LIN {X 0,Y 632.972,Z 1080.137,A -85,B 0,C 180,E1 6544.862,E2 6544.862} C_VEL
LIN {X 0,Y 629.315,Z 1123.898,A -85,B 0,C 180,E1 6550.738,E2 6550.738} C_VEL
LIN {X 0,Y 627.45,Z 1154.06,A -85,B 0,C 180,E1 6556.727,E2 6556.727} C_VEL
LIN {X 0,Y 627.035,Z 1171.451,A -85,B 0,C 180,E1 6562.357,E2 6562.357} C_VEL
LIN {X 0,Y 626.816,Z 1179.339,A -85,B 0,C 180,E1 6567.922,E2 6567.922} C_VEL
LIN {X 0,Y 626.99,Z 1178.178,A -85,B 0,C 180,E1 6573.468,E2 6573.468} C_VEL
LIN {X 0,Y 627.101,Z 1167.787,A -85,B 0,C 180,E1 6579.045,E2 6579.045} C_VEL
LIN {X 0,Y 627.936,Z 1145.964,A -85,B 0,C 180,E1 6585.071,E2 6585.071} C_VEL
LIN {X 0,Y 630.384,Z 1109.697,A -85,B 0,C 180,E1 6591.339,E2 6591.339} C_VEL
LIN {X 0,Y 634.84,Z 1059.626,A -85,B 0,C 180,E1 6597.186,E2 6597.186} C_VEL
LIN {X 0,Y 640.935,Z 997.311,A -85,B 0,C 180,E1 6602.167,E2 6602.167} C_VEL
LIN {X 0,Y 646.827,Z 930.309,A -85,B 0,C 180,E1 6605.71,E2 6605.71} C_VEL
LIN {X 0,Y 651.3,Z 859.749,A -85,B 0,C 180,E1 6607.946,E2 6607.946} C_VEL
LIN {X 0,Y 651.243,Z 808.043,A -85,B 0,C 180,E1 6608.958,E2 6608.958} C_VEL
LIN {X 0,Y 625.945,Z 762.06,A -85,B 0,C 180,E1 6612.013,E2 6612.013} C_VEL
LIN {X 0,Y 626.103,Z 762.06,A -85,B 0,C 180,E1 6620.047,E2 6620.047} C_VEL
LIN {X 0,Y 626.399,Z 762.06,A -85,B 0,C 180,E1 6628.62,E2 6628.62} C_VEL
LIN {X 0,Y 626.558,Z 762.06,A -85,B 0,C 180,E1 6637.961,E2 6637.961} C_VEL
LIN {X 0,Y 627.231,Z 762.06,A -85,B 0,C 180,E1 6646.724,E2 6646.724} C_VEL
LIN {X 0,Y 627.296,Z 762.06,A -85,B 0,C 180,E1 6656.747,E2 6656.747} C_VEL
LIN {X 0,Y 626.777,Z 762.06,A -85,B 0,C 180,E1 6666.27,E2 6666.27} C_VEL
LIN {X 0,Y 626.418,Z 762.06,A -85,B 0,C 180,E1 6674.754,E2 6674.754} C_VEL
LIN {X 0,Y 626.309,Z 762.06,A -85,B 0,C 180,E1 6682.078,E2 6682.078} C_VEL
LIN {X 0,Y 626.181,Z 762.06,A -85,B 0,C 180,E1 6690.708,E2 6690.708} C_VEL
LIN {X 0,Y 625.995,Z 762.06,A -85,B 0,C 180,E1 6698.209,E2 6698.209} C_VEL
LIN {X 0,Y 626.116,Z 762.06,A -85,B 0,C 180,E1 6703.678,E2 6703.678} C_VEL
LIN {X 0,Y 627.821,Z 770.775,A -85,B 0,C 180,E1 6704.212,E2 6704.212} C_VEL
LIN {X 0,Y 629.865,Z 783.636,A -85,B 0,C 180,E1 6704.574,E2 6704.574} C_VEL
LIN {X 0,Y 651.231,Z 823.405,A -85,B 0,C 180,E1 6706.95,E2 6706.95} C_VEL
LIN {X 0,Y 647.22,Z 901.729,A -85,B 0,C 180,E1 6708.805,E2 6708.805} C_VEL
LIN {X 0,Y 640.811,Z 974.236,A -85,B 0,C 180,E1 6711.939,E2 6711.939} C_VEL
LIN {X 0,Y 633.348,Z 1041.271,A -85,B 0,C 180,E1 6716.376,E2 6716.376} C_VEL
LIN {X 0,Y 626.505,Z 1100.933,A -85,B 0,C 180,E1 6722.094,E2 6722.094} C_VEL
LIN {X 0,Y 621.948,Z 1147.2,A -85,B 0,C 180,E1 6728.406,E2 6728.406} C_VEL
LIN {X 0,Y 619.779,Z 1179.297,A -85,B 0,C 180,E1 6734.748,E2 6734.748} C_VEL
LIN {X 0,Y 619.01,Z 1199.023,A -85,B 0,C 180,E1 6740.836,E2 6740.836} C_VEL
LIN {X 0,Y 618.831,Z 1208.374,A -85,B 0,C 180,E1 6746.486,E2 6746.486} C_VEL
LIN {X 0,Y 618.753,Z 1209.405,A -85,B 0,C 180,E1 6752.105,E2 6752.105} C_VEL
LIN {X 0,Y 618.943,Z 1202.167,A -85,B 0,C 180,E1 6757.743,E2 6757.743} C_VEL
LIN {X 0,Y 619.523,Z 1184.044,A -85,B 0,C 180,E1 6764.028,E2 6764.028} C_VEL
LIN {X 0,Y 621.435,Z 1154.124,A -85,B 0,C 180,E1 6770.425,E2 6770.425} C_VEL
LIN {X 0,Y 625.556,Z 1110.358,A -85,B 0,C 180,E1 6776.797,E2 6776.797} C_VEL
LIN {X 0,Y 632.02,Z 1052.823,A -85,B 0,C 180,E1 6782.674,E2 6782.674} C_VEL
LIN {X 0,Y 639.533,Z 985.869,A -85,B 0,C 180,E1 6787.417,E2 6787.417} C_VEL
LIN {X 0,Y 646.407,Z 914.616,A -85,B 0,C 180,E1 6790.745,E2 6790.745} C_VEL
LIN {X 0,Y 650.861,Z 841.464,A -85,B 0,C 180,E1 6792.732,E2 6792.732} C_VEL
LIN {X 0,Y 650.149,Z 816.893,A -85,B 0,C 180,E1 6793.253,E2 6793.253} C_VEL
LIN {X 0,Y 618.02,Z 762.06,A -85,B 0,C 180,E1 6796.943,E2 6796.943} C_VEL
LIN {X 0,Y 618.577,Z 762.06,A -85,B 0,C 180,E1 6805.212,E2 6805.212} C_VEL
LIN {X 0,Y 618.386,Z 762.06,A -85,B 0,C 180,E1 6814.546,E2 6814.546} C_VEL
LIN {X 0,Y 618.44,Z 762.06,A -85,B 0,C 180,E1 6823.591,E2 6823.591} C_VEL
LIN {X 0,Y 618.436,Z 762.06,A -85,B 0,C 180,E1 6832.228,E2 6832.228} C_VEL
LIN {X 0,Y 618.578,Z 762.06,A -85,B 0,C 180,E1 6839.283,E2 6839.283} C_VEL
LIN {X 0,Y 618.573,Z 762.06,A -85,B 0,C 180,E1 6846.839,E2 6846.839} C_VEL
LIN {X 0,Y 618.354,Z 762.06,A -85,B 0,C 180,E1 6854.921,E2 6854.921} C_VEL
LIN {X 0,Y 618.049,Z 762.06,A -85,B 0,C 180,E1 6863.057,E2 6863.057} C_VEL
LIN {X 0,Y 618.489,Z 762.06,A -85,B 0,C 180,E1 6871.828,E2 6871.828} C_VEL
LIN {X 0,Y 618.3,Z 762.06,A -85,B 0,C 180,E1 6880.562,E2 6880.562} C_VEL
LIN {X 0,Y 618.305,Z 763.681,A -85,B 0,C 180,E1 6887.36,E2 6887.36} C_VEL
LIN {X 0,Y 646.36,Z 813.844,A -85,B 0,C 180,E1 6890.637,E2 6890.637} C_VEL
LIN {X 0,Y 643.451,Z 889.072,A -85,B 0,C 180,E1 6892.263,E2 6892.263} C_VEL
LIN {X 0,Y 637.631,Z 960.527,A -85,B 0,C 180,E1 6895.184,E2 6895.184} C_VEL
LIN {X 0,Y 631.001,Z 1026.212,A -85,B 0,C 180,E1 6899.431,E2 6899.431} C_VEL
LIN {X 0,Y 625.13,Z 1083.1,A -85,B 0,C 180,E1 6904.88,E2 6904.88} C_VEL
LIN {X 0,Y 621.285,Z 1126.643,A -85,B 0,C 180,E1 6910.947,E2 6910.947} C_VEL
LIN {X 0,Y 619.446,Z 1155.409,A -85,B 0,C 180,E1 6916.913,E2 6916.913} C_VEL
LIN {X 0,Y 619.059,Z 1171.45,A -85,B 0,C 180,E1 6922.258,E2 6922.258} C_VEL
LIN {X 0,Y 618.82,Z 1179.339,A -85,B 0,C 180,E1 6927.895,E2 6927.895} C_VEL
LIN {X 0,Y 618.985,Z 1178.179,A -85,B 0,C 180,E1 6933.513,E2 6933.513} C_VEL
LIN {X 0,Y 619.092,Z 1165.857,A -85,B 0,C 180,E1 6939.875,E2 6939.875} C_VEL
LIN {X 0,Y 620.14,Z 1142.599,A -85,B 0,C 180,E1 6945.97,E2 6945.97} C_VEL
LIN {X 0,Y 622.856,Z 1107.043,A -85,B 0,C 180,E1 6951.985,E2 6951.985} C_VEL
LIN {X 0,Y 627.83,Z 1055.791,A -85,B 0,C 180,E1 6957.906,E2 6957.906} C_VEL
LIN {X 0,Y 634.324,Z 993.783,A -85,B 0,C 180,E1 6962.802,E2 6962.802} C_VEL
LIN {X 0,Y 640.691,Z 925.524,A -85,B 0,C 180,E1 6966.333,E2 6966.333} C_VEL
LIN {X 0,Y 645.573,Z 856.303,A -85,B 0,C 180,E1 6968.501,E2 6968.501} C_VEL
LIN {X 0,Y 645.401,Z 811.288,A -85,B 0,C 180,E1 6969.39,E2 6969.39} C_VEL
LIN {X 0,Y 617.998,Z 762.06,A -85,B 0,C 180,E1 6972.732,E2 6972.732} C_VEL
LIN {X 0,Y 618.138,Z 762.06,A -85,B 0,C 180,E1 6981.253,E2 6981.253} C_VEL
LIN {X 0,Y 618.383,Z 762.06,A -85,B 0,C 180,E1 6990.531,E2 6990.531} C_VEL
LIN {X 0,Y 618.488,Z 762.06,A -85,B 0,C 180,E1 6999.171,E2 6999.171} C_VEL
LIN {X 0,Y 619.321,Z 762.06,A -85,B 0,C 180,E1 7007.991,E2 7007.991} C_VEL
LIN {X 0,Y 619.217,Z 762.06,A -85,B 0,C 180,E1 7017.907,E2 7017.907} C_VEL
LIN {X 0,Y 618.579,Z 762.06,A -85,B 0,C 180,E1 7026.819,E2 7026.819} C_VEL
LIN {X 0,Y 618.378,Z 762.06,A -85,B 0,C 180,E1 7034.95,E2 7034.95} C_VEL
LIN {X 0,Y 618.109,Z 762.06,A -85,B 0,C 180,E1 7043.063,E2 7043.063} C_VEL
LIN {X 0,Y 618.003,Z 762.06,A -85,B 0,C 180,E1 7051.89,E2 7051.89} C_VEL
LIN {X 0,Y 617.716,Z 762.06,A -85,B 0,C 180,E1 7060.646,E2 7060.646} C_VEL
LIN {X 0,Y 618.142,Z 763.584,A -85,B 0,C 180,E1 7063.287,E2 7063.287} C_VEL
LIN {X 0,Y 629.865,Z 783.636,A -85,B 0,C 180,E1 7064.574,E2 7064.574} C_VEL
LIN {X 0,Y 640.224,Z 814.553,A -85,B 0,C 180,E1 7065.868,E2 7065.868} C_VEL
LIN {X 0,Y 645.268,Z 827.537,A -85,B 0,C 180,E1 7066.528,E2 7066.528} C_VEL
LIN {X 0,Y 640.734,Z 906.147,A -85,B 0,C 180,E1 7068.474,E2 7068.474} C_VEL
LIN {X 0,Y 633.667,Z 980.13,A -85,B 0,C 180,E1 7071.809,E2 7071.809} C_VEL
LIN {X 0,Y 625.559,Z 1048.266,A -85,B 0,C 180,E1 7076.534,E2 7076.534} C_VEL
LIN {X 0,Y 618.451,Z 1107.346,A -85,B 0,C 180,E1 7082.492,E2 7082.492} C_VEL
LIN {X 0,Y 614.002,Z 1153.543,A -85,B 0,C 180,E1 7089.215,E2 7089.215} C_VEL
LIN {X 0,Y 612.007,Z 1186.192,A -85,B 0,C 180,E1 7096.383,E2 7096.383} C_VEL
LIN {X 0,Y 611.482,Z 1204.733,A -85,B 0,C 180,E1 7103.591,E2 7103.591} C_VEL
LIN {X 0,Y 611.017,Z 1209.838,A -85,B 0,C 180,E1 7110.71,E2 7110.71} C_VEL
LIN {X 0,Y 610.986,Z 1203.526,A -85,B 0,C 180,E1 7117.128,E2 7117.128} C_VEL
LIN {X 0,Y 611.464,Z 1187.527,A -85,B 0,C 180,E1 7123.261,E2 7123.261} C_VEL
LIN {X 0,Y 613.202,Z 1159.147,A -85,B 0,C 180,E1 7129.766,E2 7129.766} C_VEL
LIN {X 0,Y 617.273,Z 1117.563,A -85,B 0,C 180,E1 7136.222,E2 7136.222} C_VEL
LIN {X 0,Y 624.02,Z 1060.465,A -85,B 0,C 180,E1 7142.405,E2 7142.405} C_VEL
LIN {X 0,Y 632.018,Z 994.245,A -85,B 0,C 180,E1 7147.364,E2 7147.364} C_VEL
LIN {X 0,Y 639.415,Z 923.76,A -85,B 0,C 180,E1 7150.864,E2 7150.864} C_VEL
LIN {X 0,Y 644.561,Z 848.588,A -85,B 0,C 180,E1 7153.084,E2 7153.084} C_VEL
LIN {X 0,Y 644.019,Z 819.648,A -85,B 0,C 180,E1 7153.719,E2 7153.719} C_VEL
LIN {X 0,Y 610.073,Z 762.06,A -85,B 0,C 180,E1 7157.493,E2 7157.493} C_VEL
LIN {X 0,Y 610.558,Z 762.06,A -85,B 0,C 180,E1 7166.31,E2 7166.31} C_VEL
LIN {X 0,Y 610.263,Z 762.06,A -85,B 0,C 180,E1 7175.095,E2 7175.095} C_VEL
LIN {X 0,Y 610.44,Z 762.06,A -85,B 0,C 180,E1 7183.37,E2 7183.37} C_VEL
LIN {X 0,Y 610.446,Z 762.06,A -85,B 0,C 180,E1 7192.125,E2 7192.125} C_VEL
LIN {X 0,Y 610.579,Z 762.06,A -85,B 0,C 180,E1 7199.273,E2 7199.273} C_VEL
LIN {X 0,Y 610.725,Z 762.06,A -85,B 0,C 180,E1 7206.406,E2 7206.406} C_VEL
LIN {X 0,Y 610.3,Z 762.06,A -85,B 0,C 180,E1 7215.122,E2 7215.122} C_VEL
LIN {X 0,Y 610.129,Z 762.06,A -85,B 0,C 180,E1 7222.665,E2 7222.665} C_VEL
LIN {X 0,Y 610.454,Z 762.06,A -85,B 0,C 180,E1 7231.015,E2 7231.015} C_VEL
LIN {X 0,Y 610.262,Z 762.06,A -85,B 0,C 180,E1 7239.343,E2 7239.343} C_VEL
LIN {X 0,Y 610.277,Z 763.855,A -85,B 0,C 180,E1 7246.599,E2 7246.599} C_VEL
LIN {X 0,Y 640.61,Z 817.11,A -85,B 0,C 180,E1 7250.202,E2 7250.202} C_VEL
LIN {X 0,Y 637.307,Z 890.904,A -85,B 0,C 180,E1 7251.834,E2 7251.834} C_VEL
LIN {X 0,Y 630.91,Z 960.513,A -85,B 0,C 180,E1 7254.758,E2 7254.758} C_VEL
LIN {X 0,Y 623.825,Z 1026.845,A -85,B 0,C 180,E1 7259.098,E2 7259.098} C_VEL
LIN {X 0,Y 617.637,Z 1083.093,A -85,B 0,C 180,E1 7264.554,E2 7264.554} C_VEL
LIN {X 0,Y 613.482,Z 1126.638,A -85,B 0,C 180,E1 7270.695,E2 7270.695} C_VEL
LIN {X 0,Y 611.529,Z 1155.408,A -85,B 0,C 180,E1 7276.74,E2 7276.74} C_VEL
LIN {X 0,Y 611.029,Z 1173.317,A -85,B 0,C 180,E1 7283.016,E2 7283.016} C_VEL
LIN {X 0,Y 610.859,Z 1179.847,A -85,B 0,C 180,E1 7289.29,E2 7289.29} C_VEL
LIN {X 0,Y 611.275,Z 1175.345,A -85,B 0,C 180,E1 7295.697,E2 7295.697} C_VEL
LIN {X 0,Y 612.229,Z 1156.406,A -85,B 0,C 180,E1 7302.883,E2 7302.883} C_VEL
LIN {X 0,Y 614.178,Z 1122.729,A -85,B 0,C 180,E1 7309.866,E2 7309.866} C_VEL
LIN {X 0,Y 618.595,Z 1076.123,A -85,B 0,C 180,E1 7316.154,E2 7316.154} C_VEL
LIN {X 0,Y 624.868,Z 1018.535,A -85,B 0,C 180,E1 7321.454,E2 7321.454} C_VEL
LIN {X 0,Y 631.781,Z 951.617,A -85,B 0,C 180,E1 7325.604,E2 7325.604} C_VEL
LIN {X 0,Y 637.934,Z 879.426,A -85,B 0,C 180,E1 7328.425,E2 7328.425} C_VEL
LIN {X 0,Y 639.65,Z 814.585,A -85,B 0,C 180,E1 7329.828,E2 7329.828} C_VEL
LIN {X 0,Y 610.11,Z 762.06,A -85,B 0,C 180,E1 7333.577,E2 7333.577} C_VEL
LIN {X 0,Y 610.17,Z 762.06,A -85,B 0,C 180,E1 7342.469,E2 7342.469} C_VEL
LIN {X 0,Y 610.341,Z 762.06,A -85,B 0,C 180,E1 7351.009,E2 7351.009} C_VEL
LIN {X 0,Y 610.46,Z 762.06,A -85,B 0,C 180,E1 7358.884,E2 7358.884} C_VEL
LIN {X 0,Y 611.247,Z 762.06,A -85,B 0,C 180,E1 7368.529,E2 7368.529} C_VEL
LIN {X 0,Y 611.236,Z 762.06,A -85,B 0,C 180,E1 7377.88,E2 7377.88} C_VEL
LIN {X 0,Y 610.707,Z 762.06,A -85,B 0,C 180,E1 7386.436,E2 7386.436} C_VEL
LIN {X 0,Y 610.321,Z 762.06,A -85,B 0,C 180,E1 7395.152,E2 7395.152} C_VEL
LIN {X 0,Y 610.181,Z 762.06,A -85,B 0,C 180,E1 7402.694,E2 7402.694} C_VEL
LIN {X 0,Y 610.098,Z 762.06,A -85,B 0,C 180,E1 7410.953,E2 7410.953} C_VEL
LIN {X 0,Y 609.786,Z 762.06,A -85,B 0,C 180,E1 7419.418,E2 7419.418} C_VEL
LIN {X 0,Y 610.156,Z 764.104,A -85,B 0,C 180,E1 7422.596,E2 7422.596} C_VEL
LIN {X 0,Y 640.224,Z 814.553,A -85,B 0,C 180,E1 7425.868,E2 7425.868} C_VEL
LIN {X 0,Y 639.91,Z 831.931,A -85,B 0,C 180,E1 7426.142,E2 7426.142} C_VEL
LIN {X 0,Y 639.001,Z 838.231,A -85,B 0,C 180,E1 7426.202,E2 7426.202} C_VEL
LIN {X 0,Y 633.48,Z 918.001,A -85,B 0,C 180,E1 7428.399,E2 7428.399} C_VEL
LIN {X 0,Y 625.961,Z 990.66,A -85,B 0,C 180,E1 7431.956,E2 7431.956} C_VEL
LIN {X 0,Y 617.597,Z 1056.725,A -85,B 0,C 180,E1 7436.844,E2 7436.844} C_VEL
LIN {X 0,Y 610.467,Z 1113.066,A -85,B 0,C 180,E1 7442.851,E2 7442.851} C_VEL
LIN {X 0,Y 605.973,Z 1157.974,A -85,B 0,C 180,E1 7449.76,E2 7449.76} C_VEL
LIN {X 0,Y 604.058,Z 1189.883,A -85,B 0,C 180,E1 7457.309,E2 7457.309} C_VEL
LIN {X 0,Y 603.382,Z 1205.908,A -85,B 0,C 180,E1 7464.249,E2 7464.249} C_VEL
LIN {X 0,Y 603.012,Z 1209.838,A -85,B 0,C 180,E1 7470.719,E2 7470.719} C_VEL
LIN {X 0,Y 602.988,Z 1203.524,A -85,B 0,C 180,E1 7477.223,E2 7477.223} C_VEL
LIN {X 0,Y 603.509,Z 1187.527,A -85,B 0,C 180,E1 7483.439,E2 7483.439} C_VEL
LIN {X 0,Y 605.336,Z 1160.03,A -85,B 0,C 180,E1 7489.861,E2 7489.861} C_VEL
LIN {X 0,Y 609.687,Z 1118.343,A -85,B 0,C 180,E1 7496.467,E2 7496.467} C_VEL
LIN {X 0,Y 616.724,Z 1062.438,A -85,B 0,C 180,E1 7502.64,E2 7502.64} C_VEL
LIN {X 0,Y 625.308,Z 995.453,A -85,B 0,C 180,E1 7507.748,E2 7507.748} C_VEL
LIN {X 0,Y 633.183,Z 924.545,A -85,B 0,C 180,E1 7511.317,E2 7511.317} C_VEL
LIN {X 0,Y 638.671,Z 849.436,A -85,B 0,C 180,E1 7513.559,E2 7513.559} C_VEL
LIN {X 0,Y 638.209,Z 823.006,A -85,B 0,C 180,E1 7514.158,E2 7514.158} C_VEL
LIN {X 0,Y 602.105,Z 762.06,A -85,B 0,C 180,E1 7518.367,E2 7518.367} C_VEL
LIN {X 0,Y 602.468,Z 762.06,A -85,B 0,C 180,E1 7527.186,E2 7527.186} C_VEL
LIN {X 0,Y 602.247,Z 762.06,A -85,B 0,C 180,E1 7535.412,E2 7535.412} C_VEL
LIN {X 0,Y 602.473,Z 762.06,A -85,B 0,C 180,E1 7543.143,E2 7543.143} C_VEL
LIN {X 0,Y 602.454,Z 762.06,A -85,B 0,C 180,E1 7552.02,E2 7552.02} C_VEL
LIN {X 0,Y 602.58,Z 762.06,A -85,B 0,C 180,E1 7559.264,E2 7559.264} C_VEL
LIN {X 0,Y 602.707,Z 762.06,A -85,B 0,C 180,E1 7566.492,E2 7566.492} C_VEL
LIN {X 0,Y 602.252,Z 762.06,A -85,B 0,C 180,E1 7575.329,E2 7575.329} C_VEL
LIN {X 0,Y 602.033,Z 762.06,A -85,B 0,C 180,E1 7583.161,E2 7583.161} C_VEL
LIN {X 0,Y 602.455,Z 762.06,A -85,B 0,C 180,E1 7591.078,E2 7591.078} C_VEL
LIN {X 0,Y 602.267,Z 762.06,A -85,B 0,C 180,E1 7599.969,E2 7599.969} C_VEL
LIN {X 0,Y 602.125,Z 762.964,A -85,B 0,C 180,E1 7605.782,E2 7605.782} C_VEL
LIN {X 0,Y 634.763,Z 820.076,A -85,B 0,C 180,E1 7609.742,E2 7609.742} C_VEL
LIN {X 0,Y 631.092,Z 894.25,A -85,B 0,C 180,E1 7611.45,E2 7611.45} C_VEL
LIN {X 0,Y 624.285,Z 962.539,A -85,B 0,C 180,E1 7614.396,E2 7614.396} C_VEL
LIN {X 0,Y 616.159,Z 1031.496,A -85,B 0,C 180,E1 7619.086,E2 7619.086} C_VEL
LIN {X 0,Y 609.691,Z 1087.332,A -85,B 0,C 180,E1 7624.72,E2 7624.72} C_VEL
LIN {X 0,Y 605.444,Z 1129.882,A -85,B 0,C 180,E1 7630.998,E2 7630.998} C_VEL
LIN {X 0,Y 603.483,Z 1158.086,A -85,B 0,C 180,E1 7637.299,E2 7637.299} C_VEL
LIN {X 0,Y 603.087,Z 1174.516,A -85,B 0,C 180,E1 7643.64,E2 7643.64} C_VEL
LIN {X 0,Y 602.857,Z 1179.847,A -85,B 0,C 180,E1 7649.281,E2 7649.281} C_VEL
LIN {X 0,Y 603.303,Z 1175.346,A -85,B 0,C 180,E1 7655.772,E2 7655.772} C_VEL
LIN {X 0,Y 604.272,Z 1156.407,A -85,B 0,C 180,E1 7663.055,E2 7663.055} C_VEL
LIN {X 0,Y 606.328,Z 1123.607,A -85,B 0,C 180,E1 7669.981,E2 7669.981} C_VEL
LIN {X 0,Y 611.098,Z 1076.452,A -85,B 0,C 180,E1 7676.463,E2 7676.463} C_VEL
LIN {X 0,Y 617.827,Z 1018.541,A -85,B 0,C 180,E1 7681.854,E2 7681.854} C_VEL
LIN {X 0,Y 625.884,Z 948.387,A -85,B 0,C 180,E1 7686.246,E2 7686.246} C_VEL
LIN {X 0,Y 632.245,Z 876.975,A -85,B 0,C 180,E1 7688.99,E2 7688.99} C_VEL
LIN {X 0,Y 633.798,Z 817.777,A -85,B 0,C 180,E1 7690.289,E2 7690.289} C_VEL
LIN {X 0,Y 602.12,Z 762.06,A -85,B 0,C 180,E1 7694.292,E2 7694.292} C_VEL
LIN {X 0,Y 602.142,Z 762.06,A -85,B 0,C 180,E1 7703.694,E2 7703.694} C_VEL
LIN {X 0,Y 602.259,Z 762.06,A -85,B 0,C 180,E1 7712.227,E2 7712.227} C_VEL
LIN {X 0,Y 602.323,Z 762.06,A -85,B 0,C 180,E1 7720.767,E2 7720.767} C_VEL
LIN {X 0,Y 603.225,Z 762.06,A -85,B 0,C 180,E1 7729.137,E2 7729.137} C_VEL
LIN {X 0,Y 603.233,Z 762.06,A -85,B 0,C 180,E1 7737.852,E2 7737.852} C_VEL
LIN {X 0,Y 602.676,Z 762.06,A -85,B 0,C 180,E1 7746.522,E2 7746.522} C_VEL
LIN {X 0,Y 602.279,Z 762.06,A -85,B 0,C 180,E1 7755.359,E2 7755.359} C_VEL
LIN {X 0,Y 602.071,Z 762.06,A -85,B 0,C 180,E1 7763.162,E2 7763.162} C_VEL
LIN {X 0,Y 602.091,Z 762.06,A -85,B 0,C 180,E1 7771.134,E2 7771.134} C_VEL
LIN {X 0,Y 601.736,Z 762.06,A -85,B 0,C 180,E1 7780.051,E2 7780.051} C_VEL
LIN {X 0,Y 601.924,Z 763.538,A -85,B 0,C 180,E1 7781.827,E2 7781.827} C_VEL
LIN {X 0,Y 639.368,Z 830.222,A -85,B 0,C 180,E1 7786.074,E2 7786.074} C_VEL
LIN {X 0,Y 639.001,Z 838.231,A -85,B 0,C 180,E1 7786.202,E2 7786.202} C_VEL
LIN {X 0,Y 631.54,Z 872.791,A -85,B 0,C 180,E1 7786.489,E2 7786.489} C_VEL
LIN {X 0,Y 624.788,Z 945.294,A -85,B 0,C 180,E1 7789.069,E2 7789.069} C_VEL
LIN {X 0,Y 615.988,Z 1016.482,A -85,B 0,C 180,E1 7793.185,E2 7793.185} C_VEL
LIN {X 0,Y 607.505,Z 1079.463,A -85,B 0,C 180,E1 7798.613,E2 7798.613} C_VEL
LIN {X 0,Y 600.829,Z 1132.474,A -85,B 0,C 180,E1 7805.188,E2 7805.188} C_VEL
LIN {X 0,Y 596.838,Z 1172.135,A -85,B 0,C 180,E1 7812.407,E2 7812.407} C_VEL
LIN {X 0,Y 595.351,Z 1195.465,A -85,B 0,C 180,E1 7819.049,E2 7819.049} C_VEL
LIN {X 0,Y 595.088,Z 1206.795,A -85,B 0,C 180,E1 7824.881,E2 7824.881} C_VEL
LIN {X 0,Y 595.032,Z 1209.838,A -85,B 0,C 180,E1 7830.729,E2 7830.729} C_VEL
LIN {X 0,Y 594.999,Z 1203.521,A -85,B 0,C 180,E1 7837.32,E2 7837.32} C_VEL
LIN {X 0,Y 595.591,Z 1186.203,A -85,B 0,C 180,E1 7843.997,E2 7843.997} C_VEL
LIN {X 0,Y 597.679,Z 1158.561,A -85,B 0,C 180,E1 7850.418,E2 7850.418} C_VEL
LIN {X 0,Y 602.303,Z 1116.951,A -85,B 0,C 180,E1 7857.009,E2 7857.009} C_VEL
LIN {X 0,Y 609.999,Z 1059.857,A -85,B 0,C 180,E1 7863.306,E2 7863.306} C_VEL
LIN {X 0,Y 619.009,Z 993.875,A -85,B 0,C 180,E1 7868.316,E2 7868.316} C_VEL
LIN {X 0,Y 627.143,Z 924.111,A -85,B 0,C 180,E1 7871.824,E2 7871.824} C_VEL
LIN {X 0,Y 632.814,Z 849.722,A -85,B 0,C 180,E1 7874.048,E2 7874.048} C_VEL
LIN {X 0,Y 632.259,Z 826.44,A -85,B 0,C 180,E1 7874.572,E2 7874.572} C_VEL
LIN {X 0,Y 594.208,Z 762.06,A -85,B 0,C 180,E1 7879.119,E2 7879.119} C_VEL
LIN {X 0,Y 594.409,Z 762.06,A -85,B 0,C 180,E1 7886.684,E2 7886.684} C_VEL
LIN {X 0,Y 594.237,Z 762.06,A -85,B 0,C 180,E1 7895.058,E2 7895.058} C_VEL
LIN {X 0,Y 594.259,Z 762.06,A -85,B 0,C 180,E1 7904.428,E2 7904.428} C_VEL
LIN {X 0,Y 594.462,Z 762.06,A -85,B 0,C 180,E1 7911.912,E2 7911.912} C_VEL
LIN {X 0,Y 594.593,Z 762.06,A -85,B 0,C 180,E1 7919.254,E2 7919.254} C_VEL
LIN {X 0,Y 594.67,Z 762.06,A -85,B 0,C 180,E1 7926.58,E2 7926.58} C_VEL
LIN {X 0,Y 594.213,Z 762.06,A -85,B 0,C 180,E1 7935.542,E2 7935.542} C_VEL
LIN {X 0,Y 594.01,Z 762.06,A -85,B 0,C 180,E1 7943.315,E2 7943.315} C_VEL
LIN {X 0,Y 594.429,Z 762.06,A -85,B 0,C 180,E1 7951.546,E2 7951.546} C_VEL
LIN {X 0,Y 594.18,Z 762.06,A -85,B 0,C 180,E1 7960.626,E2 7960.626} C_VEL
LIN {X 0,Y 594.256,Z 763.545,A -85,B 0,C 180,E1 7964.987,E2 7964.987} C_VEL
LIN {X 0,Y 629.008,Z 823.213,A -85,B 0,C 180,E1 7969.285,E2 7969.285} C_VEL
LIN {X 0,Y 625.064,Z 895.42,A -85,B 0,C 180,E1 7970.985,E2 7970.985} C_VEL
LIN {X 0,Y 617.855,Z 963.225,A -85,B 0,C 180,E1 7973.944,E2 7973.944} C_VEL
LIN {X 0,Y 609.218,Z 1030.33,A -85,B 0,C 180,E1 7978.589,E2 7978.589} C_VEL
LIN {X 0,Y 602.317,Z 1086.289,A -85,B 0,C 180,E1 7984.26,E2 7984.26} C_VEL
LIN {X 0,Y 597.641,Z 1129.879,A -85,B 0,C 180,E1 7990.74,E2 7990.74} C_VEL
LIN {X 0,Y 595.539,Z 1158.083,A -85,B 0,C 180,E1 7997.127,E2 7997.127} C_VEL
LIN {X 0,Y 595.039,Z 1174.288,A -85,B 0,C 180,E1 8003.416,E2 8003.416} C_VEL
LIN {X 0,Y 594.872,Z 1179.846,A -85,B 0,C 180,E1 8009.271,E2 8009.271} C_VEL
LIN {X 0,Y 595.331,Z 1175.399,A -85,B 0,C 180,E1 8015.819,E2 8015.819} C_VEL
LIN {X 0,Y 596.288,Z 1156.409,A -85,B 0,C 180,E1 8023.233,E2 8023.233} C_VEL
LIN {X 0,Y 598.52,Z 1123.609,A -85,B 0,C 180,E1 8030.253,E2 8030.253} C_VEL
LIN {X 0,Y 603.521,Z 1077.639,A -85,B 0,C 180,E1 8036.677,E2 8036.677} C_VEL
LIN {X 0,Y 610.673,Z 1019.813,A -85,B 0,C 180,E1 8042.167,E2 8042.167} C_VEL
LIN {X 0,Y 618.995,Z 953.671,A -85,B 0,C 180,E1 8046.473,E2 8046.473} C_VEL
LIN {X 0,Y 625.947,Z 882.027,A -85,B 0,C 180,E1 8049.353,E2 8049.353} C_VEL
LIN {X 0,Y 627.928,Z 820.81,A -85,B 0,C 180,E1 8050.766,E2 8050.766} C_VEL
LIN {X 0,Y 594.191,Z 762.06,A -85,B 0,C 180,E1 8055.133,E2 8055.133} C_VEL
LIN {X 0,Y 594.11,Z 762.06,A -85,B 0,C 180,E1 8064.931,E2 8064.931} C_VEL
LIN {X 0,Y 594.228,Z 762.06,A -85,B 0,C 180,E1 8073.466,E2 8073.466} C_VEL
LIN {X 0,Y 594.327,Z 762.06,A -85,B 0,C 180,E1 8081.4,E2 8081.4} C_VEL
LIN {X 0,Y 595.211,Z 762.06,A -85,B 0,C 180,E1 8088.989,E2 8088.989} C_VEL
LIN {X 0,Y 595.229,Z 762.06,A -85,B 0,C 180,E1 8097.823,E2 8097.823} C_VEL
LIN {X 0,Y 594.641,Z 762.06,A -85,B 0,C 180,E1 8106.611,E2 8106.611} C_VEL
LIN {X 0,Y 594.527,Z 762.06,A -85,B 0,C 180,E1 8114.051,E2 8114.051} C_VEL
LIN {X 0,Y 594.045,Z 762.06,A -85,B 0,C 180,E1 8123.347,E2 8123.347} C_VEL
LIN {X 0,Y 594.024,Z 762.06,A -85,B 0,C 180,E1 8131.605,E2 8131.605} C_VEL
LIN {X 0,Y 593.766,Z 762.06,A -85,B 0,C 180,E1 8138.83,E2 8138.83} C_VEL
LIN {X 0,Y 593.896,Z 763.614,A -85,B 0,C 180,E1 8141.039,E2 8141.039} C_VEL
LIN {X 0,Y 633.4,Z 831.798,A -85,B 0,C 180,E1 8145.61,E2 8145.61} C_VEL
LIN {X 0,Y 631.54,Z 872.791,A -85,B 0,C 180,E1 8146.489,E2 8146.489} C_VEL
LIN {X 0,Y 622.689,Z 906.696,A -85,B 0,C 180,E1 8147.015,E2 8147.015} C_VEL
LIN {X 0,Y 614.522,Z 979.053,A -85,B 0,C 180,E1 8150.32,E2 8150.32} C_VEL
LIN {X 0,Y 605.058,Z 1046.326,A -85,B 0,C 180,E1 8155.058,E2 8155.058} C_VEL
LIN {X 0,Y 596.431,Z 1105.461,A -85,B 0,C 180,E1 8161.142,E2 8161.142} C_VEL
LIN {X 0,Y 590.727,Z 1150.518,A -85,B 0,C 180,E1 8167.805,E2 8167.805} C_VEL
LIN {X 0,Y 587.977,Z 1182.006,A -85,B 0,C 180,E1 8174.626,E2 8174.626} C_VEL
LIN {X 0,Y 587.094,Z 1200.615,A -85,B 0,C 180,E1 8181.083,E2 8181.083} C_VEL
LIN {X 0,Y 587.153,Z 1209.403,A -85,B 0,C 180,E1 8187.778,E2 8187.778} C_VEL
LIN {X 0,Y 587.328,Z 1206.281,A -85,B 0,C 180,E1 8195.616,E2 8195.616} C_VEL
LIN {X 0,Y 587.539,Z 1191.036,A -85,B 0,C 180,E1 8202.672,E2 8202.672} C_VEL
LIN {X 0,Y 589.398,Z 1163.87,A -85,B 0,C 180,E1 8209.649,E2 8209.649} C_VEL
LIN {X 0,Y 594.118,Z 1123.159,A -85,B 0,C 180,E1 8216.53,E2 8216.53} C_VEL
LIN {X 0,Y 601.845,Z 1068.373,A -85,B 0,C 180,E1 8222.942,E2 8222.942} C_VEL
LIN {X 0,Y 611.221,Z 1003.832,A -85,B 0,C 180,E1 8228.159,E2 8228.159} C_VEL
LIN {X 0,Y 620.196,Z 933.124,A -85,B 0,C 180,E1 8231.963,E2 8231.963} C_VEL
LIN {X 0,Y 626.092,Z 859.422,A -85,B 0,C 180,E1 8234.324,E2 8234.324} C_VEL
LIN {X 0,Y 626.084,Z 829.765,A -85,B 0,C 180,E1 8235.002,E2 8235.002} C_VEL
LIN {X 0,Y 586.179,Z 762.06,A -85,B 0,C 180,E1 8239.796,E2 8239.796} C_VEL
LIN {X 0,Y 586.333,Z 762.06,A -85,B 0,C 180,E1 8247.931,E2 8247.931} C_VEL
LIN {X 0,Y 586.118,Z 762.06,A -85,B 0,C 180,E1 8256.707,E2 8256.707} C_VEL
LIN {X 0,Y 586.275,Z 762.06,A -85,B 0,C 180,E1 8264.211,E2 8264.211} C_VEL
LIN {X 0,Y 586.483,Z 762.06,A -85,B 0,C 180,E1 8271.801,E2 8271.801} C_VEL
LIN {X 0,Y 586.594,Z 762.06,A -85,B 0,C 180,E1 8279.244,E2 8279.244} C_VEL
LIN {X 0,Y 586.638,Z 762.06,A -85,B 0,C 180,E1 8286.671,E2 8286.671} C_VEL
LIN {X 0,Y 586.47,Z 762.06,A -85,B 0,C 180,E1 8294.217,E2 8294.217} C_VEL
LIN {X 0,Y 586.011,Z 762.06,A -85,B 0,C 180,E1 8303.269,E2 8303.269} C_VEL
LIN {X 0,Y 586.366,Z 762.06,A -85,B 0,C 180,E1 8312.031,E2 8312.031} C_VEL
LIN {X 0,Y 586.169,Z 762.06,A -85,B 0,C 180,E1 8321.302,E2 8321.302} C_VEL
LIN {X 0,Y 586.206,Z 763.284,A -85,B 0,C 180,E1 8324.126,E2 8324.126} C_VEL
LIN {X 0,Y 623.291,Z 826.304,A -85,B 0,C 180,E1 8328.818,E2 8328.818} C_VEL
LIN {X 0,Y 618.854,Z 898.927,A -85,B 0,C 180,E1 8330.587,E2 8330.587} C_VEL
LIN {X 0,Y 611.169,Z 966.822,A -85,B 0,C 180,E1 8333.651,E2 8333.651} C_VEL
LIN {X 0,Y 602.035,Z 1031.851,A -85,B 0,C 180,E1 8338.291,E2 8338.291} C_VEL
LIN {X 0,Y 594.653,Z 1087.887,A -85,B 0,C 180,E1 8344.106,E2 8344.106} C_VEL
LIN {X 0,Y 589.853,Z 1129.975,A -85,B 0,C 180,E1 8350.495,E2 8350.495} C_VEL
LIN {X 0,Y 587.602,Z 1158.08,A -85,B 0,C 180,E1 8356.95,E2 8356.95} C_VEL
LIN {X 0,Y 587.038,Z 1174.287,A -85,B 0,C 180,E1 8363.326,E2 8363.326} C_VEL
LIN {X 0,Y 586.871,Z 1179.846,A -85,B 0,C 180,E1 8369.261,E2 8369.261} C_VEL
LIN {X 0,Y 587.346,Z 1175.341,A -85,B 0,C 180,E1 8375.935,E2 8375.935} C_VEL
LIN {X 0,Y 588.301,Z 1156.411,A -85,B 0,C 180,E1 8383.416,E2 8383.416} C_VEL
LIN {X 0,Y 590.795,Z 1122.844,A -85,B 0,C 180,E1 8390.669,E2 8390.669} C_VEL
LIN {X 0,Y 596.156,Z 1076.419,A -85,B 0,C 180,E1 8397.185,E2 8397.185} C_VEL
LIN {X 0,Y 604.578,Z 1014.365,A -85,B 0,C 180,E1 8403.065,E2 8403.065} C_VEL
LIN {X 0,Y 613.379,Z 949.648,A -85,B 0,C 180,E1 8407.183,E2 8407.183} C_VEL
LIN {X 0,Y 620.384,Z 879.671,A -85,B 0,C 180,E1 8409.938,E2 8409.938} C_VEL
LIN {X 0,Y 622.12,Z 823.861,A -85,B 0,C 180,E1 8411.245,E2 8411.245} C_VEL
LIN {X 0,Y 586.081,Z 762.06,A -85,B 0,C 180,E1 8415.948,E2 8415.948} C_VEL
LIN {X 0,Y 586.095,Z 762.06,A -85,B 0,C 180,E1 8424.596,E2 8424.596} C_VEL
LIN {X 0,Y 586.194,Z 762.06,A -85,B 0,C 180,E1 8433.196,E2 8433.196} C_VEL
LIN {X 0,Y 586.298,Z 762.06,A -85,B 0,C 180,E1 8441.135,E2 8441.135} C_VEL
LIN {X 0,Y 587.241,Z 762.06,A -85,B 0,C 180,E1 8448.838,E2 8448.838} C_VEL
LIN {X 0,Y 587.224,Z 762.06,A -85,B 0,C 180,E1 8457.793,E2 8457.793} C_VEL
LIN {X 0,Y 586.627,Z 762.06,A -85,B 0,C 180,E1 8466.701,E2 8466.701} C_VEL
LIN {X 0,Y 586.473,Z 762.06,A -85,B 0,C 180,E1 8474.248,E2 8474.248} C_VEL
LIN {X 0,Y 586.061,Z 762.06,A -85,B 0,C 180,E1 8483.273,E2 8483.273} C_VEL
LIN {X 0,Y 585.937,Z 762.06,A -85,B 0,C 180,E1 8492.093,E2 8492.093} C_VEL
LIN {X 0,Y 585.758,Z 763.249,A -85,B 0,C 180,E1 8500.188,E2 8500.188} C_VEL
LIN {X 0,Y 627.244,Z 834.133,A -85,B 0,C 180,E1 8505.168,E2 8505.168} C_VEL
LIN {X 0,Y 622.689,Z 906.696,A -85,B 0,C 180,E1 8507.015,E2 8507.015} C_VEL
LIN {X 0,Y 614.028,Z 928.795,A -85,B 0,C 180,E1 8507.343,E2 8507.343} C_VEL
LIN {X 0,Y 605.269,Z 999.674,A -85,B 0,C 180,E1 8511.086,E2 8511.086} C_VEL
LIN {X 0,Y 595.428,Z 1064.977,A -85,B 0,C 180,E1 8516.303,E2 8516.303} C_VEL
LIN {X 0,Y 587.228,Z 1120.285,A -85,B 0,C 180,E1 8522.715,E2 8522.715} C_VEL
LIN {X 0,Y 582.141,Z 1163.606,A -85,B 0,C 180,E1 8530.042,E2 8530.042} C_VEL
LIN {X 0,Y 579.864,Z 1193.289,A -85,B 0,C 180,E1 8537.922,E2 8537.922} C_VEL
LIN {X 0,Y 579.164,Z 1206.789,A -85,B 0,C 180,E1 8544.74,E2 8544.74} C_VEL
LIN {X 0,Y 579.037,Z 1209.838,A -85,B 0,C 180,E1 8550.749,E2 8550.749} C_VEL
LIN {X 0,Y 579.006,Z 1203.516,A -85,B 0,C 180,E1 8557.523,E2 8557.523} C_VEL
LIN {X 0,Y 579.804,Z 1186.201,A -85,B 0,C 180,E1 8564.386,E2 8564.386} C_VEL
LIN {X 0,Y 582.454,Z 1155.592,A -85,B 0,C 180,E1 8571.576,E2 8571.576} C_VEL
LIN {X 0,Y 588.637,Z 1109.819,A -85,B 0,C 180,E1 8578.703,E2 8578.703} C_VEL
LIN {X 0,Y 597.479,Z 1051.475,A -85,B 0,C 180,E1 8584.955,E2 8584.955} C_VEL
LIN {X 0,Y 607.321,Z 985.398,A -85,B 0,C 180,E1 8589.812,E2 8589.812} C_VEL
LIN {X 0,Y 615.429,Z 918.9,A -85,B 0,C 180,E1 8593.011,E2 8593.011} C_VEL
LIN {X 0,Y 620.86,Z 846.059,A -85,B 0,C 180,E1 8595.073,E2 8595.073} C_VEL
LIN {X 0,Y 619.481,Z 832.28,A -85,B 0,C 180,E1 8595.493,E2 8595.493} C_VEL
LIN {X 0,Y 578.194,Z 762.06,A -85,B 0,C 180,E1 8600.688,E2 8600.688} C_VEL
LIN {X 0,Y 578.276,Z 762.06,A -85,B 0,C 180,E1 8609.197,E2 8609.197} C_VEL
LIN {X 0,Y 578.05,Z 762.06,A -85,B 0,C 180,E1 8617.604,E2 8617.604} C_VEL
LIN {X 0,Y 578.221,Z 762.06,A -85,B 0,C 180,E1 8625.544,E2 8625.544} C_VEL
LIN {X 0,Y 578.343,Z 762.06,A -85,B 0,C 180,E1 8633.202,E2 8633.202} C_VEL
LIN {X 0,Y 578.45,Z 762.06,A -85,B 0,C 180,E1 8640.736,E2 8640.736} C_VEL
LIN {X 0,Y 578.337,Z 762.06,A -85,B 0,C 180,E1 8648.284,E2 8648.284} C_VEL
LIN {X 0,Y 578.14,Z 762.06,A -85,B 0,C 180,E1 8656.784,E2 8656.784} C_VEL
LIN {X 0,Y 577.972,Z 762.06,A -85,B 0,C 180,E1 8665.66,E2 8665.66} C_VEL
LIN {X 0,Y 578.334,Z 762.06,A -85,B 0,C 180,E1 8674.332,E2 8674.332} C_VEL
LIN {X 0,Y 578.37,Z 764.01,A -85,B 0,C 180,E1 8683.269,E2 8683.269} C_VEL
LIN {X 0,Y 617.528,Z 829.414,A -85,B 0,C 180,E1 8688.339,E2 8688.339} C_VEL
LIN {X 0,Y 612.763,Z 901.876,A -85,B 0,C 180,E1 8690.162,E2 8690.162} C_VEL
LIN {X 0,Y 604.642,Z 969.043,A -85,B 0,C 180,E1 8693.265,E2 8693.265} C_VEL
LIN {X 0,Y 595.029,Z 1033.504,A -85,B 0,C 180,E1 8697.96,E2 8697.96} C_VEL
LIN {X 0,Y 586.554,Z 1092.338,A -85,B 0,C 180,E1 8704.339,E2 8704.339} C_VEL
LIN {X 0,Y 581.694,Z 1133.803,A -85,B 0,C 180,E1 8710.983,E2 8710.983} C_VEL
LIN {X 0,Y 579.545,Z 1160.579,A -85,B 0,C 180,E1 8717.534,E2 8717.534} C_VEL
LIN {X 0,Y 579.198,Z 1175.678,A -85,B 0,C 180,E1 8724.103,E2 8724.103} C_VEL
LIN {X 0,Y 579.469,Z 1179.824,A -85,B 0,C 180,E1 8730.751,E2 8730.751} C_VEL
LIN {X 0,Y 579.352,Z 1171.251,A -85,B 0,C 180,E1 8738.279,E2 8738.279} C_VEL
LIN {X 0,Y 580.245,Z 1150.802,A -85,B 0,C 180,E1 8745.132,E2 8745.132} C_VEL
LIN {X 0,Y 583.427,Z 1117.041,A -85,B 0,C 180,E1 8751.943,E2 8751.943} C_VEL
LIN {X 0,Y 589.685,Z 1068.827,A -85,B 0,C 180,E1 8758.411,E2 8758.411} C_VEL
LIN {X 0,Y 599.005,Z 1007.843,A -85,B 0,C 180,E1 8764.067,E2 8764.067} C_VEL
LIN {X 0,Y 608.249,Z 942.473,A -85,B 0,C 180,E1 8768.063,E2 8768.063} C_VEL
LIN {X 0,Y 615.342,Z 872.939,A -85,B 0,C 180,E1 8770.644,E2 8770.644} C_VEL
LIN {X 0,Y 616.568,Z 827.594,A -85,B 0,C 180,E1 8771.693,E2 8771.693} C_VEL
LIN {X 0,Y 578.021,Z 762.06,A -85,B 0,C 180,E1 8776.802,E2 8776.802} C_VEL
LIN {X 0,Y 578.048,Z 762.06,A -85,B 0,C 180,E1 8785.734,E2 8785.734} C_VEL
LIN {X 0,Y 578.242,Z 762.06,A -85,B 0,C 180,E1 8794.801,E2 8794.801} C_VEL
LIN {X 0,Y 578.652,Z 762.06,A -85,B 0,C 180,E1 8804.029,E2 8804.029} C_VEL
LIN {X 0,Y 578.584,Z 762.06,A -85,B 0,C 180,E1 8811.72,E2 8811.72} C_VEL
LIN {X 0,Y 578.633,Z 762.06,A -85,B 0,C 180,E1 8819.264,E2 8819.264} C_VEL
LIN {X 0,Y 578.593,Z 762.06,A -85,B 0,C 180,E1 8826.795,E2 8826.795} C_VEL
LIN {X 0,Y 578.412,Z 762.06,A -85,B 0,C 180,E1 8834.451,E2 8834.451} C_VEL
LIN {X 0,Y 578.127,Z 762.06,A -85,B 0,C 180,E1 8842.392,E2 8842.392} C_VEL
LIN {X 0,Y 577.948,Z 762.06,A -85,B 0,C 180,E1 8851.481,E2 8851.481} C_VEL
LIN {X 0,Y 577.914,Z 763.772,A -85,B 0,C 180,E1 8859.343,E2 8859.343} C_VEL
LIN {X 0,Y 621.043,Z 837.745,A -85,B 0,C 180,E1 8864.745,E2 8864.745} C_VEL
LIN {X 0,Y 615.263,Z 917.722,A -85,B 0,C 180,E1 8866.922,E2 8866.922} C_VEL
LIN {X 0,Y 614.028,Z 928.795,A -85,B 0,C 180,E1 8867.343,E2 8867.343} C_VEL
LIN {X 0,Y 604.257,Z 961.165,A -85,B 0,C 180,E1 8868.364,E2 8868.364} C_VEL
LIN {X 0,Y 594.44,Z 1027.751,A -85,B 0,C 180,E1 8872.6,E2 8872.6} C_VEL
LIN {X 0,Y 584.407,Z 1089.748,A -85,B 0,C 180,E1 8878.463,E2 8878.463} C_VEL
LIN {X 0,Y 576.91,Z 1139.778,A -85,B 0,C 180,E1 8885.316,E2 8885.316} C_VEL
LIN {X 0,Y 572.729,Z 1176.407,A -85,B 0,C 180,E1 8892.716,E2 8892.716} C_VEL
LIN {X 0,Y 571.232,Z 1198.062,A -85,B 0,C 180,E1 8899.635,E2 8899.635} C_VEL
LIN {X 0,Y 570.876,Z 1208.373,A -85,B 0,C 180,E1 8906.191,E2 8906.191} C_VEL
LIN {X 0,Y 570.819,Z 1209.405,A -85,B 0,C 180,E1 8912.282,E2 8912.282} C_VEL
LIN {X 0,Y 571.293,Z 1200.616,A -85,B 0,C 180,E1 8919.163,E2 8919.163} C_VEL
LIN {X 0,Y 573.129,Z 1177.815,A -85,B 0,C 180,E1 8926.908,E2 8926.908} C_VEL
LIN {X 0,Y 577.234,Z 1139.339,A -85,B 0,C 180,E1 8934.744,E2 8934.744} C_VEL
LIN {X 0,Y 584.721,Z 1088.293,A -85,B 0,C 180,E1 8941.699,E2 8941.699} C_VEL
LIN {X 0,Y 594.715,Z 1026.436,A -85,B 0,C 180,E1 8947.5,E2 8947.5} C_VEL
LIN {X 0,Y 604.145,Z 960.293,A -85,B 0,C 180,E1 8951.696,E2 8951.696} C_VEL
LIN {X 0,Y 612.124,Z 882.953,A -85,B 0,C 180,E1 8954.699,E2 8954.699} C_VEL
LIN {X 0,Y 613.943,Z 836.635,A -85,B 0,C 180,E1 8955.866,E2 8955.866} C_VEL
LIN {X 0,Y 570.203,Z 762.06,A -85,B 0,C 180,E1 8961.68,E2 8961.68} C_VEL
LIN {X 0,Y 570.259,Z 762.06,A -85,B 0,C 180,E1 8970.484,E2 8970.484} C_VEL
LIN {X 0,Y 570.101,Z 762.06,A -85,B 0,C 180,E1 8978.919,E2 8978.919} C_VEL
LIN {X 0,Y 570.642,Z 762.06,A -85,B 0,C 180,E1 8988.477,E2 8988.477} C_VEL
LIN {X 0,Y 571.197,Z 762.06,A -85,B 0,C 180,E1 8997.7,E2 8997.7} C_VEL
LIN {X 0,Y 570.584,Z 762.06,A -85,B 0,C 180,E1 9006.859,E2 9006.859} C_VEL
LIN {X 0,Y 570.375,Z 762.06,A -85,B 0,C 180,E1 9014.627,E2 9014.627} C_VEL
LIN {X 0,Y 569.951,Z 762.06,A -85,B 0,C 180,E1 9023.373,E2 9023.373} C_VEL
LIN {X 0,Y 570.329,Z 762.06,A -85,B 0,C 180,E1 9031.243,E2 9031.243} C_VEL
LIN {X 0,Y 570.098,Z 762.06,A -85,B 0,C 180,E1 9040.703,E2 9040.703} C_VEL
LIN {X 0,Y 570.303,Z 763.625,A -85,B 0,C 180,E1 9042.327,E2 9042.327} C_VEL
LIN {X 0,Y 611.724,Z 832.301,A -85,B 0,C 180,E1 9047.853,E2 9047.853} C_VEL
LIN {X 0,Y 606.543,Z 906.082,A -85,B 0,C 180,E1 9049.772,E2 9049.772} C_VEL
LIN {X 0,Y 598.014,Z 972.489,A -85,B 0,C 180,E1 9052.942,E2 9052.942} C_VEL
LIN {X 0,Y 587.863,Z 1036.251,A -85,B 0,C 180,E1 9057.715,E2 9057.715} C_VEL
LIN {X 0,Y 579.054,Z 1092.331,A -85,B 0,C 180,E1 9063.982,E2 9063.982} C_VEL
LIN {X 0,Y 573.894,Z 1133.798,A -85,B 0,C 180,E1 9070.714,E2 9070.714} C_VEL
LIN {X 0,Y 571.586,Z 1160.578,A -85,B 0,C 180,E1 9077.358,E2 9077.358} C_VEL
LIN {X 0,Y 571.166,Z 1175.495,A -85,B 0,C 180,E1 9083.905,E2 9083.905} C_VEL
LIN {X 0,Y 571.464,Z 1179.824,A -85,B 0,C 180,E1 9090.762,E2 9090.762} C_VEL
LIN {X 0,Y 571.447,Z 1172.821,A -85,B 0,C 180,E1 9097.627,E2 9097.627} C_VEL
LIN {X 0,Y 572.301,Z 1152.257,A -85,B 0,C 180,E1 9104.974,E2 9104.974} C_VEL
LIN {X 0,Y 575.6,Z 1118.248,A -85,B 0,C 180,E1 9112.053,E2 9112.053} C_VEL
LIN {X 0,Y 582.445,Z 1069.181,A -85,B 0,C 180,E1 9118.797,E2 9118.797} C_VEL
LIN {X 0,Y 592.242,Z 1009.582,A -85,B 0,C 180,E1 9124.442,E2 9124.442} C_VEL
LIN {X 0,Y 602.102,Z 944.039,A -85,B 0,C 180,E1 9128.522,E2 9128.522} C_VEL
LIN {X 0,Y 609.415,Z 875.354,A -85,B 0,C 180,E1 9131.115,E2 9131.115} C_VEL
LIN {X 0,Y 610.651,Z 830.421,A -85,B 0,C 180,E1 9132.192,E2 9132.192} C_VEL
LIN {X 0,Y 569.952,Z 762.06,A -85,B 0,C 180,E1 9137.736,E2 9137.736} C_VEL
LIN {X 0,Y 570.049,Z 762.06,A -85,B 0,C 180,E1 9146.937,E2 9146.937} C_VEL
LIN {X 0,Y 570.265,Z 762.06,A -85,B 0,C 180,E1 9156.562,E2 9156.562} C_VEL
LIN {X 0,Y 571.114,Z 762.06,A -85,B 0,C 180,E1 9166.96,E2 9166.96} C_VEL
LIN {X 0,Y 571.223,Z 762.06,A -85,B 0,C 180,E1 9177.731,E2 9177.731} C_VEL
LIN {X 0,Y 570.579,Z 762.06,A -85,B 0,C 180,E1 9186.891,E2 9186.891} C_VEL
LIN {X 0,Y 570.366,Z 762.06,A -85,B 0,C 180,E1 9194.66,E2 9194.66} C_VEL
LIN {X 0,Y 569.974,Z 762.06,A -85,B 0,C 180,E1 9203.371,E2 9203.371} C_VEL
LIN {X 0,Y 569.968,Z 762.06,A -85,B 0,C 180,E1 9211.302,E2 9211.302} C_VEL
LIN {X 0,Y 569.97,Z 763.952,A -85,B 0,C 180,E1 9218.438,E2 9218.438} C_VEL
LIN {X 0,Y 614.875,Z 840.193,A -85,B 0,C 180,E1 9224.296,E2 9224.296} C_VEL
LIN {X 0,Y 608.68,Z 920.385,A -85,B 0,C 180,E1 9226.545,E2 9226.545} C_VEL
LIN {X 0,Y 604.257,Z 961.165,A -85,B 0,C 180,E1 9228.364,E2 9228.364} C_VEL
LIN {X 0,Y 593.568,Z 992.304,A -85,B 0,C 180,E1 9229.632,E2 9229.632} C_VEL
LIN {X 0,Y 583.032,Z 1056.111,A -85,B 0,C 180,E1 9234.529,E2 9234.529} C_VEL
LIN {X 0,Y 573.181,Z 1113.794,A -85,B 0,C 180,E1 9241.031,E2 9241.031} C_VEL
LIN {X 0,Y 566.848,Z 1157.115,A -85,B 0,C 180,E1 9248.114,E2 9248.114} C_VEL
LIN {X 0,Y 564.118,Z 1187.281,A -85,B 0,C 180,E1 9255.527,E2 9255.527} C_VEL
LIN {X 0,Y 563.474,Z 1204.716,A -85,B 0,C 180,E1 9263.042,E2 9263.042} C_VEL
LIN {X 0,Y 563.041,Z 1209.838,A -85,B 0,C 180,E1 9270.77,E2 9270.77} C_VEL
LIN {X 0,Y 563.044,Z 1203.51,A -85,B 0,C 180,E1 9277.738,E2 9277.738} C_VEL
LIN {X 0,Y 563.97,Z 1186.199,A -85,B 0,C 180,E1 9284.799,E2 9284.799} C_VEL
LIN {X 0,Y 567.206,Z 1155.134,A -85,B 0,C 180,E1 9292.282,E2 9292.282} C_VEL
LIN {X 0,Y 574.254,Z 1108.444,A -85,B 0,C 180,E1 9299.678,E2 9299.678} C_VEL
LIN {X 0,Y 583.965,Z 1051.058,A -85,B 0,C 180,E1 9305.929,E2 9305.929} C_VEL
LIN {X 0,Y 594.338,Z 986.705,A -85,B 0,C 180,E1 9310.718,E2 9310.718} C_VEL
LIN {X 0,Y 603.535,Z 913.278,A -85,B 0,C 180,E1 9314.193,E2 9314.193} C_VEL
LIN {X 0,Y 607.62,Z 839.601,A -85,B 0,C 180,E1 9316.326,E2 9316.326} C_VEL
LIN {X 0,Y 562.225,Z 762.06,A -85,B 0,C 180,E1 9322.72,E2 9322.72} C_VEL
LIN {X 0,Y 562.246,Z 762.06,A -85,B 0,C 180,E1 9331.791,E2 9331.791} C_VEL
LIN {X 0,Y 562.369,Z 762.06,A -85,B 0,C 180,E1 9341.901,E2 9341.901} C_VEL
LIN {X 0,Y 562.5,Z 762.06,A -85,B 0,C 180,E1 9351.449,E2 9351.449} C_VEL
LIN {X 0,Y 562.625,Z 762.06,A -85,B 0,C 180,E1 9359.211,E2 9359.211} C_VEL
LIN {X 0,Y 562.553,Z 762.06,A -85,B 0,C 180,E1 9366.958,E2 9366.958} C_VEL
LIN {X 0,Y 562.316,Z 762.06,A -85,B 0,C 180,E1 9374.842,E2 9374.842} C_VEL
LIN {X 0,Y 561.995,Z 762.06,A -85,B 0,C 180,E1 9383.037,E2 9383.037} C_VEL
LIN {X 0,Y 562.276,Z 762.06,A -85,B 0,C 180,E1 9391.836,E2 9391.836} C_VEL
LIN {X 0,Y 562.207,Z 763.118,A -85,B 0,C 180,E1 9401.334,E2 9401.334} C_VEL
LIN {X 0,Y 606.051,Z 835.524,A -85,B 0,C 180,E1 9407.379,E2 9407.379} C_VEL
LIN {X 0,Y 600.467,Z 908.563,A -85,B 0,C 180,E1 9409.325,E2 9409.325} C_VEL
LIN {X 0,Y 591.451,Z 975.472,A -85,B 0,C 180,E1 9412.58,E2 9412.58} C_VEL
LIN {X 0,Y 580.681,Z 1039.109,A -85,B 0,C 180,E1 9417.48,E2 9417.48} C_VEL
LIN {X 0,Y 571.375,Z 1093.986,A -85,B 0,C 180,E1 9423.83,E2 9423.83} C_VEL
LIN {X 0,Y 565.904,Z 1135.748,A -85,B 0,C 180,E1 9430.837,E2 9430.837} C_VEL
LIN {X 0,Y 563.578,Z 1162.875,A -85,B 0,C 180,E1 9437.965,E2 9437.965} C_VEL
LIN {X 0,Y 563.308,Z 1176.569,A -85,B 0,C 180,E1 9444.595,E2 9444.595} C_VEL
LIN {X 0,Y 563.214,Z 1179.271,A -85,B 0,C 180,E1 9452.316,E2 9452.316} C_VEL
LIN {X 0,Y 563.246,Z 1169.684,A -85,B 0,C 180,E1 9459.298,E2 9459.298} C_VEL
LIN {X 0,Y 564.505,Z 1149.189,A -85,B 0,C 180,E1 9465.985,E2 9465.985} C_VEL
LIN {X 0,Y 568.383,Z 1114.887,A -85,B 0,C 180,E1 9472.926,E2 9472.926} C_VEL
LIN {X 0,Y 576.367,Z 1063.78,A -85,B 0,C 180,E1 9479.889,E2 9479.889} C_VEL
LIN {X 0,Y 586.874,Z 1002.855,A -85,B 0,C 180,E1 9485.472,E2 9485.472} C_VEL
LIN {X 0,Y 596.862,Z 938.468,A -85,B 0,C 180,E1 9489.324,E2 9489.324} C_VEL
LIN {X 0,Y 604.214,Z 869.034,A -85,B 0,C 180,E1 9491.799,E2 9491.799} C_VEL
LIN {X 0,Y 604.909,Z 833.707,A -85,B 0,C 180,E1 9492.673,E2 9492.673} C_VEL
LIN {X 0,Y 561.951,Z 762.06,A -85,B 0,C 180,E1 9498.815,E2 9498.815} C_VEL
LIN {X 0,Y 562.092,Z 762.06,A -85,B 0,C 180,E1 9508.246,E2 9508.246} C_VEL
LIN {X 0,Y 562.306,Z 762.06,A -85,B 0,C 180,E1 9516.976,E2 9516.976} C_VEL
LIN {X 0,Y 563.1,Z 762.06,A -85,B 0,C 180,E1 9526.771,E2 9526.771} C_VEL
LIN {X 0,Y 563.215,Z 762.06,A -85,B 0,C 180,E1 9537.699,E2 9537.699} C_VEL
LIN {X 0,Y 562.547,Z 762.06,A -85,B 0,C 180,E1 9546.99,E2 9546.99} C_VEL
LIN {X 0,Y 562.309,Z 762.06,A -85,B 0,C 180,E1 9554.875,E2 9554.875} C_VEL
LIN {X 0,Y 562.003,Z 762.06,A -85,B 0,C 180,E1 9563.071,E2 9563.071} C_VEL
LIN {X 0,Y 561.894,Z 762.06,A -85,B 0,C 180,E1 9571.804,E2 9571.804} C_VEL
LIN {X 0,Y 562.002,Z 764.012,A -85,B 0,C 180,E1 9577.483,E2 9577.483} C_VEL
LIN {X 0,Y 606.227,Z 838.676,A -85,B 0,C 180,E1 9583.533,E2 9583.533} C_VEL
LIN {X 0,Y 608.363,Z 849.563,A -85,B 0,C 180,E1 9583.981,E2 9583.981} C_VEL
LIN {X 0,Y 601.404,Z 929.052,A -85,B 0,C 180,E1 9586.392,E2 9586.392} C_VEL
LIN {X 0,Y 593.568,Z 992.304,A -85,B 0,C 180,E1 9589.632,E2 9589.632} C_VEL
LIN {X 0,Y 582.214,Z 1022.047,A -85,B 0,C 180,E1 9591.164,E2 9591.164} C_VEL
LIN {X 0,Y 571.548,Z 1082.967,A -85,B 0,C 180,E1 9596.802,E2 9596.802} C_VEL
LIN {X 0,Y 562.872,Z 1134.912,A -85,B 0,C 180,E1 9603.796,E2 9603.796} C_VEL
LIN {X 0,Y 557.415,Z 1174.676,A -85,B 0,C 180,E1 9611.766,E2 9611.766} C_VEL
LIN {X 0,Y 555.416,Z 1197.213,A -85,B 0,C 180,E1 9618.98,E2 9618.98} C_VEL
LIN {X 0,Y 554.907,Z 1208.372,A -85,B 0,C 180,E1 9626.081,E2 9626.081} C_VEL
LIN {X 0,Y 554.85,Z 1209.405,A -85,B 0,C 180,E1 9632.348,E2 9632.348} C_VEL
LIN {X 0,Y 555.39,Z 1200.61,A -85,B 0,C 180,E1 9639.428,E2 9639.428} C_VEL
LIN {X 0,Y 557.327,Z 1177.728,A -85,B 0,C 180,E1 9647.425,E2 9647.425} C_VEL
LIN {X 0,Y 562.028,Z 1139.057,A -85,B 0,C 180,E1 9655.51,E2 9655.51} C_VEL
LIN {X 0,Y 570.458,Z 1088.44,A -85,B 0,C 180,E1 9662.568,E2 9662.568} C_VEL
LIN {X 0,Y 581.37,Z 1027.658,A -85,B 0,C 180,E1 9668.396,E2 9668.396} C_VEL
LIN {X 0,Y 591.89,Z 956.341,A -85,B 0,C 180,E1 9672.852,E2 9672.852} C_VEL
LIN {X 0,Y 600.223,Z 878.707,A -85,B 0,C 180,E1 9675.826,E2 9675.826} C_VEL
LIN {X 0,Y 601.731,Z 843.417,A -85,B 0,C 180,E1 9676.739,E2 9676.739} C_VEL
LIN {X 0,Y 557.225,Z 768.323,A -85,B 0,C 180,E1 9683.03,E2 9683.03} C_VEL
LIN {X 0,Y 554.192,Z 762.06,A -85,B 0,C 180,E1 9683.825,E2 9683.825} C_VEL
LIN {X 0,Y 554.183,Z 762.06,A -85,B 0,C 180,E1 9693.116,E2 9693.116} C_VEL
LIN {X 0,Y 554.318,Z 762.06,A -85,B 0,C 180,E1 9701.629,E2 9701.629} C_VEL
LIN {X 0,Y 554.524,Z 762.06,A -85,B 0,C 180,E1 9711.325,E2 9711.325} C_VEL
LIN {X 0,Y 554.626,Z 762.06,A -85,B 0,C 180,E1 9719.2,E2 9719.2} C_VEL
LIN {X 0,Y 554.547,Z 762.06,A -85,B 0,C 180,E1 9727.059,E2 9727.059} C_VEL
LIN {X 0,Y 554.272,Z 762.06,A -85,B 0,C 180,E1 9735.062,E2 9735.062} C_VEL
LIN {X 0,Y 553.915,Z 762.06,A -85,B 0,C 180,E1 9743.489,E2 9743.489} C_VEL
LIN {X 0,Y 554.236,Z 762.06,A -85,B 0,C 180,E1 9752.258,E2 9752.258} C_VEL
LIN {X 0,Y 554.218,Z 763.567,A -85,B 0,C 180,E1 9760.322,E2 9760.322} C_VEL
LIN {X 0,Y 600.225,Z 838.422,A -85,B 0,C 180,E1 9766.875,E2 9766.875} C_VEL
LIN {X 0,Y 594.276,Z 911.671,A -85,B 0,C 180,E1 9768.901,E2 9768.901} C_VEL
LIN {X 0,Y 584.888,Z 978.596,A -85,B 0,C 180,E1 9772.228,E2 9772.228} C_VEL
LIN {X 0,Y 573.618,Z 1041.3,A -85,B 0,C 180,E1 9777.184,E2 9777.184} C_VEL
LIN {X 0,Y 563.804,Z 1095.842,A -85,B 0,C 180,E1 9783.654,E2 9783.654} C_VEL
LIN {X 0,Y 557.936,Z 1137.697,A -85,B 0,C 180,E1 9790.965,E2 9790.965} C_VEL
LIN {X 0,Y 555.61,Z 1164.023,A -85,B 0,C 180,E1 9798.189,E2 9798.189} C_VEL
LIN {X 0,Y 555.288,Z 1176.568,A -85,B 0,C 180,E1 9804.517,E2 9804.517} C_VEL
LIN {X 0,Y 555.204,Z 1179.272,A -85,B 0,C 180,E1 9812.35,E2 9812.35} C_VEL
LIN {X 0,Y 555.245,Z 1169.685,A -85,B 0,C 180,E1 9819.433,E2 9819.433} C_VEL
LIN {X 0,Y 556.631,Z 1149.19,A -85,B 0,C 180,E1 9826.217,E2 9826.217} C_VEL
LIN {X 0,Y 560.799,Z 1114.979,A -85,B 0,C 180,E1 9833.254,E2 9833.254} C_VEL
LIN {X 0,Y 569.239,Z 1065.016,A -85,B 0,C 180,E1 9840.24,E2 9840.24} C_VEL
LIN {X 0,Y 580.379,Z 1004.07,A -85,B 0,C 180,E1 9845.921,E2 9845.921} C_VEL
LIN {X 0,Y 590.649,Z 940.303,A -85,B 0,C 180,E1 9849.777,E2 9849.777} C_VEL
LIN {X 0,Y 598.38,Z 870.606,A -85,B 0,C 180,E1 9852.3,E2 9852.3} C_VEL
LIN {X 0,Y 599.171,Z 836.943,A -85,B 0,C 180,E1 9853.166,E2 9853.166} C_VEL
LIN {X 0,Y 556.624,Z 768.06,A -85,B 0,C 180,E1 9859.179,E2 9859.179} C_VEL
LIN {X 0,Y 553.891,Z 762.06,A -85,B 0,C 180,E1 9859.933,E2 9859.933} C_VEL
LIN {X 0,Y 554.1,Z 762.06,A -85,B 0,C 180,E1 9869.571,E2 9869.571} C_VEL
LIN {X 0,Y 554.278,Z 762.06,A -85,B 0,C 180,E1 9878.322,E2 9878.322} C_VEL
LIN {X 0,Y 555.165,Z 762.06,A -85,B 0,C 180,E1 9888.184,E2 9888.184} C_VEL
LIN {X 0,Y 555.206,Z 762.06,A -85,B 0,C 180,E1 9897.666,E2 9897.666} C_VEL
LIN {X 0,Y 554.545,Z 762.06,A -85,B 0,C 180,E1 9907.091,E2 9907.091} C_VEL
LIN {X 0,Y 554.276,Z 762.06,A -85,B 0,C 180,E1 9915.095,E2 9915.095} C_VEL
LIN {X 0,Y 553.949,Z 762.06,A -85,B 0,C 180,E1 9923.489,E2 9923.489} C_VEL
LIN {X 0,Y 553.807,Z 762.06,A -85,B 0,C 180,E1 9932.324,E2 9932.324} C_VEL
LIN {X 0,Y 553.991,Z 763.949,A -85,B 0,C 180,E1 9936.471,E2 9936.471} C_VEL
LIN {X 0,Y 596.668,Z 835.186,A -85,B 0,C 180,E1 9942.605,E2 9942.605} C_VEL
LIN {X 0,Y 602.348,Z 850.683,A -85,B 0,C 180,E1 9943.497,E2 9943.497} C_VEL
LIN {X 0,Y 594.966,Z 930.71,A -85,B 0,C 180,E1 9945.963,E2 9945.963} C_VEL
LIN {X 0,Y 585.013,Z 1004.934,A -85,B 0,C 180,E1 9949.964,E2 9949.964} C_VEL
LIN {X 0,Y 582.214,Z 1022.047,A -85,B 0,C 180,E1 9951.164,E2 9951.164} C_VEL
LIN {X 0,Y 570.647,Z 1050.086,A -85,B 0,C 180,E1 9953.001,E2 9953.001} C_VEL
LIN {X 0,Y 559.698,Z 1107.681,A -85,B 0,C 180,E1 9959.362,E2 9959.362} C_VEL
LIN {X 0,Y 552.098,Z 1152.367,A -85,B 0,C 180,E1 9966.527,E2 9966.527} C_VEL
LIN {X 0,Y 548.346,Z 1183.506,A -85,B 0,C 180,E1 9973.943,E2 9973.943} C_VEL
LIN {X 0,Y 547.17,Z 1202.16,A -85,B 0,C 180,E1 9981.23,E2 9981.23} C_VEL
LIN {X 0,Y 547.561,Z 1209.837,A -85,B 0,C 180,E1 9989.205,E2 9989.205} C_VEL
LIN {X 0,Y 547.093,Z 1204.715,A -85,B 0,C 180,E1 9997.164,E2 9997.164} C_VEL
LIN {X 0,Y 547.869,Z 1188.959,A -85,B 0,C 180,E1 10004.34,E2 10004.34} C_VEL
LIN {X 0,Y 550.934,Z 1160.501,A -85,B 0,C 180,E1 10011.813,E2 10011.813} C_VEL
LIN {X 0,Y 557.815,Z 1118.223,A -85,B 0,C 180,E1 10019.168,E2 10019.168} C_VEL
LIN {X 0,Y 568.46,Z 1061.348,A -85,B 0,C 180,E1 10025.935,E2 10025.935} C_VEL
LIN {X 0,Y 579.701,Z 996.271,A -85,B 0,C 180,E1 10031.069,E2 10031.069} C_VEL
LIN {X 0,Y 589.804,Z 924.571,A -85,B 0,C 180,E1 10034.749,E2 10034.749} C_VEL
LIN {X 0,Y 595.582,Z 846.864,A -85,B 0,C 180,E1 10037.194,E2 10037.194} C_VEL
LIN {X 0,Y 553.26,Z 774.479,A -85,B 0,C 180,E1 10043.408,E2 10043.408} C_VEL
LIN {X 0,Y 546.184,Z 762.06,A -85,B 0,C 180,E1 10044.832,E2 10044.832} C_VEL
LIN {X 0,Y 546.098,Z 762.06,A -85,B 0,C 180,E1 10054.488,E2 10054.488} C_VEL
LIN {X 0,Y 546.294,Z 762.06,A -85,B 0,C 180,E1 10063.274,E2 10063.274} C_VEL
LIN {X 0,Y 546.524,Z 762.06,A -85,B 0,C 180,E1 10071.197,E2 10071.197} C_VEL
LIN {X 0,Y 546.641,Z 762.06,A -85,B 0,C 180,E1 10079.188,E2 10079.188} C_VEL
LIN {X 0,Y 546.52,Z 762.06,A -85,B 0,C 180,E1 10087.163,E2 10087.163} C_VEL
LIN {X 0,Y 546.223,Z 762.06,A -85,B 0,C 180,E1 10095.289,E2 10095.289} C_VEL
LIN {X 0,Y 545.894,Z 762.06,A -85,B 0,C 180,E1 10103.758,E2 10103.758} C_VEL
LIN {X 0,Y 546.21,Z 762.06,A -85,B 0,C 180,E1 10112.791,E2 10112.791} C_VEL
LIN {X 0,Y 546.209,Z 763.921,A -85,B 0,C 180,E1 10119.253,E2 10119.253} C_VEL
LIN {X 0,Y 592.674,Z 838.113,A -85,B 0,C 180,E1 10126.121,E2 10126.121} C_VEL
LIN {X 0,Y 593.924,Z 850.655,A -85,B 0,C 180,E1 10126.571,E2 10126.571} C_VEL
LIN {X 0,Y 586.814,Z 923.972,A -85,B 0,C 180,E1 10128.846,E2 10128.846} C_VEL
LIN {X 0,Y 576.486,Z 991.636,A -85,B 0,C 180,E1 10132.552,E2 10132.552} C_VEL
LIN {X 0,Y 564.856,Z 1052.568,A -85,B 0,C 180,E1 10137.795,E2 10137.795} C_VEL
LIN {X 0,Y 554.983,Z 1104.842,A -85,B 0,C 180,E1 10144.572,E2 10144.572} C_VEL
LIN {X 0,Y 549.598,Z 1146.297,A -85,B 0,C 180,E1 10152.703,E2 10152.703} C_VEL
LIN {X 0,Y 547.706,Z 1169.873,A -85,B 0,C 180,E1 10160.439,E2 10160.439} C_VEL
LIN {X 0,Y 546.903,Z 1179.336,A -85,B 0,C 180,E1 10167.618,E2 10167.618} C_VEL
LIN {X 0,Y 547.044,Z 1178.187,A -85,B 0,C 180,E1 10173.976,E2 10173.976} C_VEL
LIN {X 0,Y 547.776,Z 1164.9,A -85,B 0,C 180,E1 10181.58,E2 10181.58} C_VEL
LIN {X 0,Y 550.645,Z 1137.252,A -85,B 0,C 180,E1 10189.3,E2 10189.3} C_VEL
LIN {X 0,Y 557.255,Z 1093.605,A -85,B 0,C 180,E1 10197.018,E2 10197.018} C_VEL
LIN {X 0,Y 567.405,Z 1040.171,A -85,B 0,C 180,E1 10203.357,E2 10203.357} C_VEL
LIN {X 0,Y 578.619,Z 978.576,A -85,B 0,C 180,E1 10208.234,E2 10208.234} C_VEL
LIN {X 0,Y 588.672,Z 908.632,A -85,B 0,C 180,E1 10211.677,E2 10211.677} C_VEL
LIN {X 0,Y 593.554,Z 840.561,A -85,B 0,C 180,E1 10213.637,E2 10213.637} C_VEL
LIN {X 0,Y 552.428,Z 773.826,A -85,B 0,C 180,E1 10219.61,E2 10219.61} C_VEL
LIN {X 0,Y 545.845,Z 762.06,A -85,B 0,C 180,E1 10220.957,E2 10220.957} C_VEL
LIN {X 0,Y 546.071,Z 762.06,A -85,B 0,C 180,E1 10230.914,E2 10230.914} C_VEL
LIN {X 0,Y 546.226,Z 762.06,A -85,B 0,C 180,E1 10239.693,E2 10239.693} C_VEL
LIN {X 0,Y 547.149,Z 762.06,A -85,B 0,C 180,E1 10248.008,E2 10248.008} C_VEL
LIN {X 0,Y 547.205,Z 762.06,A -85,B 0,C 180,E1 10257.632,E2 10257.632} C_VEL
LIN {X 0,Y 546.514,Z 762.06,A -85,B 0,C 180,E1 10267.196,E2 10267.196} C_VEL
LIN {X 0,Y 546.225,Z 762.06,A -85,B 0,C 180,E1 10275.323,E2 10275.323} C_VEL
LIN {X 0,Y 545.927,Z 762.06,A -85,B 0,C 180,E1 10283.792,E2 10283.792} C_VEL
LIN {X 0,Y 545.766,Z 762.06,A -85,B 0,C 180,E1 10292.86,E2 10292.86} C_VEL
LIN {X 0,Y 545.855,Z 763.547,A -85,B 0,C 180,E1 10295.378,E2 10295.378} C_VEL
LIN {X 0,Y 585.206,Z 828.83,A -85,B 0,C 180,E1 10301.363,E2 10301.363} C_VEL
LIN {X 0,Y 596.327,Z 852.495,A -85,B 0,C 180,E1 10303.016,E2 10303.016} C_VEL
LIN {X 0,Y 588.538,Z 932.354,A -85,B 0,C 180,E1 10305.532,E2 10305.532} C_VEL
LIN {X 0,Y 578.34,Z 1005.175,A -85,B 0,C 180,E1 10309.508,E2 10309.508} C_VEL
LIN {X 0,Y 570.647,Z 1050.086,A -85,B 0,C 180,E1 10313.001,E2 10313.001} C_VEL
LIN {X 0,Y 560.454,Z 1068.019,A -85,B 0,C 180,E1 10314.244,E2 10314.244} C_VEL
LIN {X 0,Y 549.73,Z 1123.149,A -85,B 0,C 180,E1 10321.132,E2 10321.132} C_VEL
LIN {X 0,Y 542.914,Z 1166.173,A -85,B 0,C 180,E1 10329.135,E2 10329.135} C_VEL
LIN {X 0,Y 540.206,Z 1193.287,A -85,B 0,C 180,E1 10337.02,E2 10337.02} C_VEL
LIN {X 0,Y 539.286,Z 1206.775,A -85,B 0,C 180,E1 10344.35,E2 10344.35} C_VEL
LIN {X 0,Y 539.028,Z 1209.837,A -85,B 0,C 180,E1 10350.804,E2 10350.804} C_VEL
LIN {X 0,Y 539.102,Z 1203.501,A -85,B 0,C 180,E1 10358.084,E2 10358.084} C_VEL
LIN {X 0,Y 540.561,Z 1184.857,A -85,B 0,C 180,E1 10365.873,E2 10365.873} C_VEL
LIN {X 0,Y 545.385,Z 1150.307,A -85,B 0,C 180,E1 10374.191,E2 10374.191} C_VEL
LIN {X 0,Y 553.684,Z 1102.836,A -85,B 0,C 180,E1 10381.701,E2 10381.701} C_VEL
LIN {X 0,Y 563.997,Z 1048.604,A -85,B 0,C 180,E1 10387.577,E2 10387.577} C_VEL
LIN {X 0,Y 575.64,Z 980.455,A -85,B 0,C 180,E1 10392.529,E2 10392.529} C_VEL
LIN {X 0,Y 585.757,Z 905.97,A -85,B 0,C 180,E1 10395.967,E2 10395.967} C_VEL
LIN {X 0,Y 589.458,Z 850.12,A -85,B 0,C 180,E1 10397.678,E2 10397.678} C_VEL
LIN {X 0,Y 549.383,Z 780.601,A -85,B 0,C 180,E1 10403.785,E2 10403.785} C_VEL
LIN {X 0,Y 538.161,Z 762.06,A -85,B 0,C 180,E1 10405.886,E2 10405.886} C_VEL
LIN {X 0,Y 538.074,Z 762.06,A -85,B 0,C 180,E1 10414.055,E2 10414.055} C_VEL
LIN {X 0,Y 538.242,Z 762.06,A -85,B 0,C 180,E1 10422.76,E2 10422.76} C_VEL
LIN {X 0,Y 538.541,Z 762.06,A -85,B 0,C 180,E1 10431.066,E2 10431.066} C_VEL
LIN {X 0,Y 538.657,Z 762.06,A -85,B 0,C 180,E1 10439.176,E2 10439.176} C_VEL
LIN {X 0,Y 538.493,Z 762.06,A -85,B 0,C 180,E1 10447.27,E2 10447.27} C_VEL
LIN {X 0,Y 538.192,Z 762.06,A -85,B 0,C 180,E1 10455.523,E2 10455.523} C_VEL
LIN {X 0,Y 537.856,Z 762.06,A -85,B 0,C 180,E1 10464.135,E2 10464.135} C_VEL
LIN {X 0,Y 538.122,Z 762.06,A -85,B 0,C 180,E1 10473.765,E2 10473.765} C_VEL
LIN {X 0,Y 538.237,Z 763.928,A -85,B 0,C 180,E1 10478.122,E2 10478.122} C_VEL
LIN {X 0,Y 580.999,Z 831.275,A -85,B 0,C 180,E1 10484.77,E2 10484.77} C_VEL
LIN {X 0,Y 588.561,Z 847.688,A -85,B 0,C 180,E1 10485.954,E2 10485.954} C_VEL
LIN {X 0,Y 581.334,Z 921.196,A -85,B 0,C 180,E1 10488.18,E2 10488.18} C_VEL
LIN {X 0,Y 570.788,Z 988.581,A -85,B 0,C 180,E1 10491.805,E2 10491.805} C_VEL
LIN {X 0,Y 558.98,Z 1048.277,A -85,B 0,C 180,E1 10496.815,E2 10496.815} C_VEL
LIN {X 0,Y 548.492,Z 1100.81,A -85,B 0,C 180,E1 10503.465,E2 10503.465} C_VEL
LIN {X 0,Y 542.143,Z 1139.63,A -85,B 0,C 180,E1 10510.813,E2 10510.813} C_VEL
LIN {X 0,Y 539.691,Z 1165.129,A -85,B 0,C 180,E1 10518.247,E2 10518.247} C_VEL
LIN {X 0,Y 539.303,Z 1178.286,A -85,B 0,C 180,E1 10525.97,E2 10525.97} C_VEL
LIN {X 0,Y 539.183,Z 1179.211,A -85,B 0,C 180,E1 10532.514,E2 10532.514} C_VEL
LIN {X 0,Y 539.307,Z 1170.044,A -85,B 0,C 180,E1 10539.529,E2 10539.529} C_VEL
LIN {X 0,Y 540.931,Z 1149.193,A -85,B 0,C 180,E1 10546.702,E2 10546.702} C_VEL
LIN {X 0,Y 546.247,Z 1113.24,A -85,B 0,C 180,E1 10554.393,E2 10554.393} C_VEL
LIN {X 0,Y 555.941,Z 1063.323,A -85,B 0,C 180,E1 10561.448,E2 10561.448} C_VEL
LIN {X 0,Y 567.708,Z 1004.826,A -85,B 0,C 180,E1 10566.946,E2 10566.946} C_VEL
LIN {X 0,Y 578.868,Z 939.35,A -85,B 0,C 180,E1 10570.918,E2 10570.918} C_VEL
LIN {X 0,Y 587.136,Z 869.923,A -85,B 0,C 180,E1 10573.421,E2 10573.421} C_VEL
LIN {X 0,Y 587.598,Z 843.814,A -85,B 0,C 180,E1 10574.154,E2 10574.154} C_VEL
LIN {X 0,Y 548.31,Z 779.442,A -85,B 0,C 180,E1 10580.045,E2 10580.045} C_VEL
LIN {X 0,Y 537.816,Z 762.06,A -85,B 0,C 180,E1 10582.184,E2 10582.184} C_VEL
LIN {X 0,Y 538.012,Z 762.06,A -85,B 0,C 180,E1 10590.435,E2 10590.435} C_VEL
LIN {X 0,Y 538.216,Z 762.06,A -85,B 0,C 180,E1 10599.377,E2 10599.377} C_VEL
LIN {X 0,Y 539.112,Z 762.06,A -85,B 0,C 180,E1 10607.827,E2 10607.827} C_VEL
LIN {X 0,Y 539.194,Z 762.06,A -85,B 0,C 180,E1 10617.597,E2 10617.597} C_VEL
LIN {X 0,Y 538.485,Z 762.06,A -85,B 0,C 180,E1 10627.304,E2 10627.304} C_VEL
LIN {X 0,Y 538.203,Z 762.06,A -85,B 0,C 180,E1 10635.557,E2 10635.557} C_VEL
LIN {X 0,Y 537.899,Z 762.06,A -85,B 0,C 180,E1 10644.17,E2 10644.17} C_VEL
LIN {X 0,Y 537.671,Z 762.06,A -85,B 0,C 180,E1 10653.687,E2 10653.687} C_VEL
LIN {X 0,Y 538.068,Z 764.538,A -85,B 0,C 180,E1 10654.305,E2 10654.305} C_VEL
LIN {X 0,Y 575.318,Z 824.195,A -85,B 0,C 180,E1 10660.226,E2 10660.226} C_VEL
LIN {X 0,Y 590.253,Z 856.17,A -85,B 0,C 180,E1 10662.566,E2 10662.566} C_VEL
LIN {X 0,Y 581.889,Z 935.427,A -85,B 0,C 180,E1 10665.161,E2 10665.161} C_VEL
LIN {X 0,Y 571.098,Z 1008.553,A -85,B 0,C 180,E1 10669.263,E2 10669.263} C_VEL
LIN {X 0,Y 560.454,Z 1068.019,A -85,B 0,C 180,E1 10674.244,E2 10674.244} C_VEL
LIN {X 0,Y 548.562,Z 1092.889,A -85,B 0,C 180,E1 10676.563,E2 10676.563} C_VEL
LIN {X 0,Y 538.95,Z 1142.279,A -85,B 0,C 180,E1 10683.916,E2 10683.916} C_VEL
LIN {X 0,Y 533.458,Z 1177.749,A -85,B 0,C 180,E1 10691.776,E2 10691.776} C_VEL
LIN {X 0,Y 531.392,Z 1199.025,A -85,B 0,C 180,E1 10699.308,E2 10699.308} C_VEL
LIN {X 0,Y 530.943,Z 1208.372,A -85,B 0,C 180,E1 10705.904,E2 10705.904} C_VEL
LIN {X 0,Y 530.881,Z 1209.405,A -85,B 0,C 180,E1 10712.454,E2 10712.454} C_VEL
LIN {X 0,Y 531.493,Z 1200.778,A -85,B 0,C 180,E1 10719.762,E2 10719.762} C_VEL
LIN {X 0,Y 533.591,Z 1177.622,A -85,B 0,C 180,E1 10728.255,E2 10728.255} C_VEL
LIN {X 0,Y 539.195,Z 1139.887,A -85,B 0,C 180,E1 10736.517,E2 10736.517} C_VEL
LIN {X 0,Y 549.137,Z 1089.433,A -85,B 0,C 180,E1 10743.862,E2 10743.862} C_VEL
LIN {X 0,Y 561.073,Z 1027.648,A -85,B 0,C 180,E1 10749.801,E2 10749.801} C_VEL
LIN {X 0,Y 572.755,Z 957.276,A -85,B 0,C 180,E1 10754.302,E2 10754.302} C_VEL
LIN {X 0,Y 582.501,Z 878.063,A -85,B 0,C 180,E1 10757.425,E2 10757.425} C_VEL
LIN {X 0,Y 583.447,Z 853.397,A -85,B 0,C 180,E1 10758.178,E2 10758.178} C_VEL
LIN {X 0,Y 545.539,Z 786.659,A -85,B 0,C 180,E1 10764.167,E2 10764.167} C_VEL
LIN {X 0,Y 530.11,Z 762.06,A -85,B 0,C 180,E1 10767.225,E2 10767.225} C_VEL
LIN {X 0,Y 529.962,Z 762.06,A -85,B 0,C 180,E1 10775.445,E2 10775.445} C_VEL
LIN {X 0,Y 530.177,Z 762.06,A -85,B 0,C 180,E1 10784.201,E2 10784.201} C_VEL
LIN {X 0,Y 530.362,Z 762.06,A -85,B 0,C 180,E1 10792.584,E2 10792.584} C_VEL
LIN {X 0,Y 530.679,Z 762.06,A -85,B 0,C 180,E1 10799.164,E2 10799.164} C_VEL
LIN {X 0,Y 530.47,Z 762.06,A -85,B 0,C 180,E1 10807.381,E2 10807.381} C_VEL
LIN {X 0,Y 530.097,Z 762.06,A -85,B 0,C 180,E1 10816.595,E2 10816.595} C_VEL
LIN {X 0,Y 529.861,Z 762.06,A -85,B 0,C 180,E1 10826.341,E2 10826.341} C_VEL
LIN {X 0,Y 530.045,Z 762.06,A -85,B 0,C 180,E1 10835.925,E2 10835.925} C_VEL
LIN {X 0,Y 530.314,Z 764.143,A -85,B 0,C 180,E1 10836.94,E2 10836.94} C_VEL
LIN {X 0,Y 569.579,Z 824.98,A -85,B 0,C 180,E1 10843.373,E2 10843.373} C_VEL
LIN {X 0,Y 582.742,Z 851.589,A -85,B 0,C 180,E1 10845.458,E2 10845.458} C_VEL
LIN {X 0,Y 574.94,Z 925.633,A -85,B 0,C 180,E1 10847.797,E2 10847.797} C_VEL
LIN {X 0,Y 563.652,Z 993.896,A -85,B 0,C 180,E1 10851.614,E2 10851.614} C_VEL
LIN {X 0,Y 551.364,Z 1053.401,A -85,B 0,C 180,E1 10856.811,E2 10856.811} C_VEL
LIN {X 0,Y 540.471,Z 1104.572,A -85,B 0,C 180,E1 10863.601,E2 10863.601} C_VEL
LIN {X 0,Y 534.104,Z 1143.077,A -85,B 0,C 180,E1 10871.297,E2 10871.297} C_VEL
LIN {X 0,Y 531.826,Z 1168.02,A -85,B 0,C 180,E1 10879.32,E2 10879.32} C_VEL
LIN {X 0,Y 531.295,Z 1178.285,A -85,B 0,C 180,E1 10885.91,E2 10885.91} C_VEL
LIN {X 0,Y 531.227,Z 1179.272,A -85,B 0,C 180,E1 10892.456,E2 10892.456} C_VEL
LIN {X 0,Y 531.308,Z 1169.725,A -85,B 0,C 180,E1 10899.844,E2 10899.844} C_VEL
LIN {X 0,Y 533.526,Z 1146.792,A -85,B 0,C 180,E1 10907.686,E2 10907.686} C_VEL
LIN {X 0,Y 539.84,Z 1108.85,A -85,B 0,C 180,E1 10915.591,E2 10915.591} C_VEL
LIN {X 0,Y 550.537,Z 1057.306,A -85,B 0,C 180,E1 10922.657,E2 10922.657} C_VEL
LIN {X 0,Y 562.78,Z 997.992,A -85,B 0,C 180,E1 10927.997,E2 10927.997} C_VEL
LIN {X 0,Y 574.314,Z 930.674,A -85,B 0,C 180,E1 10931.881,E2 10931.881} C_VEL
LIN {X 0,Y 582.227,Z 862.074,A -85,B 0,C 180,E1 10934.183,E2 10934.183} C_VEL
LIN {X 0,Y 581.607,Z 846.88,A -85,B 0,C 180,E1 10934.694,E2 10934.694} C_VEL
LIN {X 0,Y 542.517,Z 781.931,A -85,B 0,C 180,E1 10940.786,E2 10940.786} C_VEL
LIN {X 0,Y 529.856,Z 762.06,A -85,B 0,C 180,E1 10943.141,E2 10943.141} C_VEL
LIN {X 0,Y 529.997,Z 762.06,A -85,B 0,C 180,E1 10951.821,E2 10951.821} C_VEL
LIN {X 0,Y 530.222,Z 762.06,A -85,B 0,C 180,E1 10960.798,E2 10960.798} C_VEL
LIN {X 0,Y 530.975,Z 762.06,A -85,B 0,C 180,E1 10969.309,E2 10969.309} C_VEL
LIN {X 0,Y 530.681,Z 762.06,A -85,B 0,C 180,E1 10979.197,E2 10979.197} C_VEL
LIN {X 0,Y 530.459,Z 762.06,A -85,B 0,C 180,E1 10987.415,E2 10987.415} C_VEL
LIN {X 0,Y 530.08,Z 762.06,A -85,B 0,C 180,E1 10996.578,E2 10996.578} C_VEL
LIN {X 0,Y 529.856,Z 762.06,A -85,B 0,C 180,E1 11006.379,E2 11006.379} C_VEL
LIN {X 0,Y 529.909,Z 764.015,A -85,B 0,C 180,E1 11013.077,E2 11013.077} C_VEL
LIN {X 0,Y 567.178,Z 822.993,A -85,B 0,C 180,E1 11019.295,E2 11019.295} C_VEL
LIN {X 0,Y 584.281,Z 859.646,A -85,B 0,C 180,E1 11022.107,E2 11022.107} C_VEL
LIN {X 0,Y 575.165,Z 939.486,A -85,B 0,C 180,E1 11024.831,E2 11024.831} C_VEL
LIN {X 0,Y 563.759,Z 1012.551,A -85,B 0,C 180,E1 11029.064,E2 11029.064} C_VEL
LIN {X 0,Y 551.81,Z 1076.182,A -85,B 0,C 180,E1 11034.665,E2 11034.665} C_VEL
LIN {X 0,Y 548.562,Z 1092.889,A -85,B 0,C 180,E1 11036.563,E2 11036.563} C_VEL
LIN {X 0,Y 536.473,Z 1115.655,A -85,B 0,C 180,E1 11039.139,E2 11039.139} C_VEL
LIN {X 0,Y 528.091,Z 1159.354,A -85,B 0,C 180,E1 11046.929,E2 11046.929} C_VEL
LIN {X 0,Y 524.275,Z 1188.702,A -85,B 0,C 180,E1 11054.908,E2 11054.908} C_VEL
LIN {X 0,Y 523.431,Z 1205.879,A -85,B 0,C 180,E1 11063.343,E2 11063.343} C_VEL
LIN {X 0,Y 523.037,Z 1209.837,A -85,B 0,C 180,E1 11070.829,E2 11070.829} C_VEL
LIN {X 0,Y 523.152,Z 1203.495,A -85,B 0,C 180,E1 11078.332,E2 11078.332} C_VEL
LIN {X 0,Y 524.895,Z 1184.856,A -85,B 0,C 180,E1 11086.36,E2 11086.36} C_VEL
LIN {X 0,Y 530.081,Z 1150.913,A -85,B 0,C 180,E1 11094.81,E2 11094.81} C_VEL
LIN {X 0,Y 539.268,Z 1103.562,A -85,B 0,C 180,E1 11102.527,E2 11102.527} C_VEL
LIN {X 0,Y 551.166,Z 1044.158,A -85,B 0,C 180,E1 11108.903,E2 11108.903} C_VEL
LIN {X 0,Y 563.515,Z 975.461,A -85,B 0,C 180,E1 11113.838,E2 11113.838} C_VEL
LIN {X 0,Y 574.66,Z 899,A -85,B 0,C 180,E1 11117.309,E2 11117.309} C_VEL
LIN {X 0,Y 577.602,Z 857.155,A -85,B 0,C 180,E1 11118.651,E2 11118.651} C_VEL
LIN {X 0,Y 542.233,Z 793.348,A -85,B 0,C 180,E1 11124.471,E2 11124.471} C_VEL
LIN {X 0,Y 522.102,Z 762.06,A -85,B 0,C 180,E1 11128.245,E2 11128.245} C_VEL
LIN {X 0,Y 521.908,Z 762.06,A -85,B 0,C 180,E1 11136.865,E2 11136.865} C_VEL
LIN {X 0,Y 522.248,Z 762.06,A -85,B 0,C 180,E1 11146.593,E2 11146.593} C_VEL
LIN {X 0,Y 522.917,Z 762.06,A -85,B 0,C 180,E1 11155.822,E2 11155.822} C_VEL
LIN {X 0,Y 522.831,Z 762.06,A -85,B 0,C 180,E1 11165.815,E2 11165.815} C_VEL
LIN {X 0,Y 522.35,Z 762.06,A -85,B 0,C 180,E1 11174.282,E2 11174.282} C_VEL
LIN {X 0,Y 521.802,Z 762.06,A -85,B 0,C 180,E1 11183.73,E2 11183.73} C_VEL
LIN {X 0,Y 522.078,Z 762.06,A -85,B 0,C 180,E1 11192.516,E2 11192.516} C_VEL
LIN {X 0,Y 522.307,Z 764.009,A -85,B 0,C 180,E1 11195.66,E2 11195.66} C_VEL
LIN {X 0,Y 560.802,Z 822.925,A -85,B 0,C 180,E1 11202.296,E2 11202.296} C_VEL
LIN {X 0,Y 577.18,Z 852.78,A -85,B 0,C 180,E1 11204.902,E2 11204.902} C_VEL
LIN {X 0,Y 569.034,Z 926.768,A -85,B 0,C 180,E1 11207.272,E2 11207.272} C_VEL
LIN {X 0,Y 557.313,Z 994.608,A -85,B 0,C 180,E1 11211.106,E2 11211.106} C_VEL
LIN {X 0,Y 544.323,Z 1055.006,A -85,B 0,C 180,E1 11216.457,E2 11216.457} C_VEL
LIN {X 0,Y 533.235,Z 1104.864,A -85,B 0,C 180,E1 11223.163,E2 11223.163} C_VEL
LIN {X 0,Y 526.301,Z 1143.323,A -85,B 0,C 180,E1 11230.974,E2 11230.974} C_VEL
LIN {X 0,Y 523.811,Z 1168.091,A -85,B 0,C 180,E1 11239.155,E2 11239.155} C_VEL
LIN {X 0,Y 523.311,Z 1178.285,A -85,B 0,C 180,E1 11245.847,E2 11245.847} C_VEL
LIN {X 0,Y 523.217,Z 1179.272,A -85,B 0,C 180,E1 11252.493,E2 11252.493} C_VEL
LIN {X 0,Y 523.33,Z 1169.726,A -85,B 0,C 180,E1 11259.995,E2 11259.995} C_VEL
LIN {X 0,Y 525.763,Z 1147.153,A -85,B 0,C 180,E1 11267.956,E2 11267.956} C_VEL
LIN {X 0,Y 532.549,Z 1108.945,A -85,B 0,C 180,E1 11276.054,E2 11276.054} C_VEL
LIN {X 0,Y 543.388,Z 1059.239,A -85,B 0,C 180,E1 11282.973,E2 11282.973} C_VEL
LIN {X 0,Y 556.208,Z 999.654,A -85,B 0,C 180,E1 11288.43,E2 11288.43} C_VEL
LIN {X 0,Y 568.236,Z 932.484,A -85,B 0,C 180,E1 11292.369,E2 11292.369} C_VEL
LIN {X 0,Y 576.564,Z 863.821,A -85,B 0,C 180,E1 11294.718,E2 11294.718} C_VEL
LIN {X 0,Y 575.868,Z 850.229,A -85,B 0,C 180,E1 11295.215,E2 11295.215} C_VEL
LIN {X 0,Y 538.585,Z 787.92,A -85,B 0,C 180,E1 11301.216,E2 11301.216} C_VEL
LIN {X 0,Y 521.885,Z 762.06,A -85,B 0,C 180,E1 11304.439,E2 11304.439} C_VEL
LIN {X 0,Y 521.96,Z 762.06,A -85,B 0,C 180,E1 11313.229,E2 11313.229} C_VEL
LIN {X 0,Y 522.29,Z 762.06,A -85,B 0,C 180,E1 11322.252,E2 11322.252} C_VEL
LIN {X 0,Y 522.7,Z 762.06,A -85,B 0,C 180,E1 11330.827,E2 11330.827} C_VEL
LIN {X 0,Y 522.684,Z 762.06,A -85,B 0,C 180,E1 11339.185,E2 11339.185} C_VEL
LIN {X 0,Y 522.452,Z 762.06,A -85,B 0,C 180,E1 11347.529,E2 11347.529} C_VEL
LIN {X 0,Y 522.121,Z 762.06,A -85,B 0,C 180,E1 11356.049,E2 11356.049} C_VEL
LIN {X 0,Y 521.822,Z 762.06,A -85,B 0,C 180,E1 11364.964,E2 11364.964} C_VEL
LIN {X 0,Y 521.83,Z 763.454,A -85,B 0,C 180,E1 11371.78,E2 11371.78} C_VEL
LIN {X 0,Y 559.835,Z 823.212,A -85,B 0,C 180,E1 11378.444,E2 11378.444} C_VEL
LIN {X 0,Y 578.478,Z 861.722,A -85,B 0,C 180,E1 11381.597,E2 11381.597} C_VEL
LIN {X 0,Y 568.959,Z 940.176,A -85,B 0,C 180,E1 11384.327,E2 11384.327} C_VEL
LIN {X 0,Y 556.842,Z 1014.136,A -85,B 0,C 180,E1 11388.688,E2 11388.688} C_VEL
LIN {X 0,Y 544.394,Z 1077.842,A -85,B 0,C 180,E1 11394.401,E2 11394.401} C_VEL
LIN {X 0,Y 536.473,Z 1115.655,A -85,B 0,C 180,E1 11399.139,E2 11399.139} C_VEL
LIN {X 0,Y 525.197,Z 1136.273,A -85,B 0,C 180,E1 11402.018,E2 11402.018} C_VEL
LIN {X 0,Y 518.501,Z 1174.676,A -85,B 0,C 180,E1 11410.343,E2 11410.343} C_VEL
LIN {X 0,Y 515.506,Z 1199.022,A -85,B 0,C 180,E1 11418.975,E2 11418.975} C_VEL
LIN {X 0,Y 514.972,Z 1208.368,A -85,B 0,C 180,E1 11425.776,E2 11425.776} C_VEL
LIN {X 0,Y 514.888,Z 1209.403,A -85,B 0,C 180,E1 11432.53,E2 11432.53} C_VEL
LIN {X 0,Y 515.579,Z 1200.595,A -85,B 0,C 180,E1 11440.163,E2 11440.163} C_VEL
LIN {X 0,Y 517.78,Z 1177.759,A -85,B 0,C 180,E1 11448.793,E2 11448.793} C_VEL
LIN {X 0,Y 523.891,Z 1141.521,A -85,B 0,C 180,E1 11457.038,E2 11457.038} C_VEL
LIN {X 0,Y 533.487,Z 1096.06,A -85,B 0,C 180,E1 11463.922,E2 11463.922} C_VEL
LIN {X 0,Y 546.144,Z 1035.511,A -85,B 0,C 180,E1 11470.134,E2 11470.134} C_VEL
LIN {X 0,Y 559.212,Z 964.379,A -85,B 0,C 180,E1 11474.997,E2 11474.997} C_VEL
LIN {X 0,Y 570.259,Z 886.427,A -85,B 0,C 180,E1 11478.306,E2 11478.306} C_VEL
LIN {X 0,Y 571.511,Z 860.265,A -85,B 0,C 180,E1 11479.181,E2 11479.181} C_VEL
LIN {X 0,Y 538.187,Z 799.043,A -85,B 0,C 180,E1 11484.907,E2 11484.907} C_VEL
LIN {X 0,Y 514.058,Z 762.06,A -85,B 0,C 180,E1 11489.72,E2 11489.72} C_VEL
LIN {X 0,Y 514.068,Z 762.06,A -85,B 0,C 180,E1 11500.133,E2 11500.133} C_VEL
LIN {X 0,Y 514.542,Z 762.06,A -85,B 0,C 180,E1 11508.928,E2 11508.928} C_VEL
LIN {X 0,Y 515.163,Z 762.06,A -85,B 0,C 180,E1 11517.45,E2 11517.45} C_VEL
LIN {X 0,Y 514.795,Z 762.06,A -85,B 0,C 180,E1 11525.906,E2 11525.906} C_VEL
LIN {X 0,Y 514.291,Z 762.06,A -85,B 0,C 180,E1 11534.51,E2 11534.51} C_VEL
LIN {X 0,Y 513.821,Z 762.06,A -85,B 0,C 180,E1 11543.483,E2 11543.483} C_VEL
LIN {X 0,Y 514.06,Z 762.06,A -85,B 0,C 180,E1 11553.088,E2 11553.088} C_VEL
LIN {X 0,Y 514.328,Z 764.032,A -85,B 0,C 180,E1 11554.303,E2 11554.303} C_VEL
LIN {X 0,Y 552.976,Z 822.229,A -85,B 0,C 180,E1 11561.313,E2 11561.313} C_VEL
LIN {X 0,Y 571.39,Z 857.95,A -85,B 0,C 180,E1 11564.423,E2 11564.423} C_VEL
LIN {X 0,Y 562.638,Z 930.952,A -85,B 0,C 180,E1 11566.873,E2 11566.873} C_VEL
LIN {X 0,Y 550.584,Z 997.277,A -85,B 0,C 180,E1 11570.737,E2 11570.737} C_VEL
LIN {X 0,Y 537.232,Z 1056.763,A -85,B 0,C 180,E1 11576.118,E2 11576.118} C_VEL
LIN {X 0,Y 525.637,Z 1106.739,A -85,B 0,C 180,E1 11582.975,E2 11582.975} C_VEL
LIN {X 0,Y 518.478,Z 1144.16,A -85,B 0,C 180,E1 11590.79,E2 11590.79} C_VEL
LIN {X 0,Y 515.816,Z 1168.309,A -85,B 0,C 180,E1 11598.985,E2 11598.985} C_VEL
LIN {X 0,Y 515.301,Z 1178.302,A -85,B 0,C 180,E1 11605.782,E2 11605.782} C_VEL
LIN {X 0,Y 515.207,Z 1179.316,A -85,B 0,C 180,E1 11612.532,E2 11612.532} C_VEL
LIN {X 0,Y 515.38,Z 1170.101,A -85,B 0,C 180,E1 11620.085,E2 11620.085} C_VEL
LIN {X 0,Y 518.137,Z 1147.153,A -85,B 0,C 180,E1 11628.341,E2 11628.341} C_VEL
LIN {X 0,Y 525.435,Z 1108.75,A -85,B 0,C 180,E1 11636.576,E2 11636.576} C_VEL
LIN {X 0,Y 536.624,Z 1059.488,A -85,B 0,C 180,E1 11643.478,E2 11643.478} C_VEL
LIN {X 0,Y 549.997,Z 999.6,A -85,B 0,C 180,E1 11649.003,E2 11649.003} C_VEL
LIN {X 0,Y 562.466,Z 932.534,A -85,B 0,C 180,E1 11652.95,E2 11652.95} C_VEL
LIN {X 0,Y 571.171,Z 862.996,A -85,B 0,C 180,E1 11655.329,E2 11655.329} C_VEL
LIN {X 0,Y 569.679,Z 852.683,A -85,B 0,C 180,E1 11655.827,E2 11655.827} C_VEL
LIN {X 0,Y 534.183,Z 793.101,A -85,B 0,C 180,E1 11661.741,E2 11661.741} C_VEL
LIN {X 0,Y 513.873,Z 762.06,A -85,B 0,C 180,E1 11665.755,E2 11665.755} C_VEL
LIN {X 0,Y 513.973,Z 762.06,A -85,B 0,C 180,E1 11674.666,E2 11674.666} C_VEL
LIN {X 0,Y 514.477,Z 762.06,A -85,B 0,C 180,E1 11683.742,E2 11683.742} C_VEL
LIN {X 0,Y 514.435,Z 762.06,A -85,B 0,C 180,E1 11692.388,E2 11692.388} C_VEL
LIN {X 0,Y 514.685,Z 762.06,A -85,B 0,C 180,E1 11699.172,E2 11699.172} C_VEL
LIN {X 0,Y 514.428,Z 762.06,A -85,B 0,C 180,E1 11707.647,E2 11707.647} C_VEL
LIN {X 0,Y 514.052,Z 762.06,A -85,B 0,C 180,E1 11716.501,E2 11716.501} C_VEL
LIN {X 0,Y 513.766,Z 762.06,A -85,B 0,C 180,E1 11725.801,E2 11725.801} C_VEL
LIN {X 0,Y 513.989,Z 764.047,A -85,B 0,C 180,E1 11730.466,E2 11730.466} C_VEL
LIN {X 0,Y 550.591,Z 820.068,A -85,B 0,C 180,E1 11737.231,E2 11737.231} C_VEL
LIN {X 0,Y 572.611,Z 865.105,A -85,B 0,C 180,E1 11741.108,E2 11741.108} C_VEL
LIN {X 0,Y 562.585,Z 943.077,A -85,B 0,C 180,E1 11743.908,E2 11743.908} C_VEL
LIN {X 0,Y 549.668,Z 1017.301,A -85,B 0,C 180,E1 11748.419,E2 11748.419} C_VEL
LIN {X 0,Y 536.929,Z 1079.858,A -85,B 0,C 180,E1 11754.171,E2 11754.171} C_VEL
LIN {X 0,Y 526.17,Z 1131.125,A -85,B 0,C 180,E1 11761.132,E2 11761.132} C_VEL
LIN {X 0,Y 525.197,Z 1136.273,A -85,B 0,C 180,E1 11762.018,E2 11762.018} C_VEL
LIN {X 0,Y 513.714,Z 1154.588,A -85,B 0,C 180,E1 11765.134,E2 11765.134} C_VEL
LIN {X 0,Y 508.855,Z 1184.381,A -85,B 0,C 180,E1 11772.953,E2 11772.953} C_VEL
LIN {X 0,Y 507.214,Z 1202.152,A -85,B 0,C 180,E1 11780.533,E2 11780.533} C_VEL
LIN {X 0,Y 507.12,Z 1209.398,A -85,B 0,C 180,E1 11787.427,E2 11787.427} C_VEL
LIN {X 0,Y 507.296,Z 1206.768,A -85,B 0,C 180,E1 11796.004,E2 11796.004} C_VEL
LIN {X 0,Y 507.924,Z 1192.521,A -85,B 0,C 180,E1 11804.118,E2 11804.118} C_VEL
LIN {X 0,Y 511.515,Z 1166.271,A -85,B 0,C 180,E1 11812.183,E2 11812.183} C_VEL
LIN {X 0,Y 519.407,Z 1126.95,A -85,B 0,C 180,E1 11819.965,E2 11819.965} C_VEL
LIN {X 0,Y 531.173,Z 1073.351,A -85,B 0,C 180,E1 11827.004,E2 11827.004} C_VEL
LIN {X 0,Y 545.111,Z 1007.328,A -85,B 0,C 180,E1 11832.831,E2 11832.831} C_VEL
LIN {X 0,Y 558.104,Z 936.304,A -85,B 0,C 180,E1 11836.955,E2 11836.955} C_VEL
LIN {X 0,Y 565.859,Z 864.252,A -85,B 0,C 180,E1 11839.65,E2 11839.65} C_VEL
LIN {X 0,Y 534.437,Z 805.033,A -85,B 0,C 180,E1 11845.305,E2 11845.305} C_VEL
LIN {X 0,Y 506,Z 762.06,A -85,B 0,C 180,E1 11851.271,E2 11851.271} C_VEL
LIN {X 0,Y 506.117,Z 762.06,A -85,B 0,C 180,E1 11861.627,E2 11861.627} C_VEL
LIN {X 0,Y 506.507,Z 762.06,A -85,B 0,C 180,E1 11870.496,E2 11870.496} C_VEL
LIN {X 0,Y 506.702,Z 762.06,A -85,B 0,C 180,E1 11879.124,E2 11879.124} C_VEL
LIN {X 0,Y 506.426,Z 762.06,A -85,B 0,C 180,E1 11887.733,E2 11887.733} C_VEL
LIN {X 0,Y 506.06,Z 762.06,A -85,B 0,C 180,E1 11896.536,E2 11896.536} C_VEL
LIN {X 0,Y 505.77,Z 762.06,A -85,B 0,C 180,E1 11905.775,E2 11905.775} C_VEL
LIN {X 0,Y 506.233,Z 763.668,A -85,B 0,C 180,E1 11912.819,E2 11912.819} C_VEL
LIN {X 0,Y 544.63,Z 820.874,A -85,B 0,C 180,E1 11920.196,E2 11920.196} C_VEL
LIN {X 0,Y 565.735,Z 860.618,A -85,B 0,C 180,E1 11923.887,E2 11923.887} C_VEL
LIN {X 0,Y 556.466,Z 933.688,A -85,B 0,C 180,E1 11926.404,E2 11926.404} C_VEL
LIN {X 0,Y 543.484,Z 1001.403,A -85,B 0,C 180,E1 11930.465,E2 11930.465} C_VEL
LIN {X 0,Y 529.256,Z 1062.013,A -85,B 0,C 180,E1 11936.172,E2 11936.172} C_VEL
LIN {X 0,Y 517.388,Z 1111.735,A -85,B 0,C 180,E1 11943.329,E2 11943.329} C_VEL
LIN {X 0,Y 510.416,Z 1147.845,A -85,B 0,C 180,E1 11951.375,E2 11951.375} C_VEL
LIN {X 0,Y 507.806,Z 1171.083,A -85,B 0,C 180,E1 11960.081,E2 11960.081} C_VEL
LIN {X 0,Y 506.966,Z 1179.582,A -85,B 0,C 180,E1 11967.43,E2 11967.43} C_VEL
LIN {X 0,Y 507.09,Z 1178.472,A -85,B 0,C 180,E1 11974.289,E2 11974.289} C_VEL
LIN {X 0,Y 508.278,Z 1165.592,A -85,B 0,C 180,E1 11982.494,E2 11982.494} C_VEL
LIN {X 0,Y 512.336,Z 1137.059,A -85,B 0,C 180,E1 11991.312,E2 11991.312} C_VEL
LIN {X 0,Y 521.354,Z 1095.014,A -85,B 0,C 180,E1 11999.324,E2 11999.324} C_VEL
LIN {X 0,Y 533.952,Z 1043.056,A -85,B 0,C 180,E1 12005.79,E2 12005.79} C_VEL
LIN {X 0,Y 547.738,Z 980.92,A -85,B 0,C 180,E1 12010.896,E2 12010.896} C_VEL
LIN {X 0,Y 559.911,Z 911.137,A -85,B 0,C 180,E1 12014.467,E2 12014.467} C_VEL
LIN {X 0,Y 565.009,Z 858.065,A -85,B 0,C 180,E1 12016.191,E2 12016.191} C_VEL
LIN {X 0,Y 530.865,Z 799.622,A -85,B 0,C 180,E1 12022.091,E2 12022.091} C_VEL
LIN {X 0,Y 505.909,Z 762.06,A -85,B 0,C 180,E1 12027.345,E2 12027.345} C_VEL
LIN {X 0,Y 506.019,Z 762.06,A -85,B 0,C 180,E1 12036.132,E2 12036.132} C_VEL
LIN {X 0,Y 506.883,Z 762.06,A -85,B 0,C 180,E1 12046.502,E2 12046.502} C_VEL
LIN {X 0,Y 507.187,Z 762.06,A -85,B 0,C 180,E1 12057.445,E2 12057.445} C_VEL
LIN {X 0,Y 506.74,Z 762.06,A -85,B 0,C 180,E1 12066.035,E2 12066.035} C_VEL
LIN {X 0,Y 506.234,Z 762.06,A -85,B 0,C 180,E1 12074.783,E2 12074.783} C_VEL
LIN {X 0,Y 505.802,Z 762.06,A -85,B 0,C 180,E1 12083.917,E2 12083.917} C_VEL
LIN {X 0,Y 505.981,Z 763.924,A -85,B 0,C 180,E1 12089.009,E2 12089.009} C_VEL
LIN {X 0,Y 542.229,Z 818.44,A -85,B 0,C 180,E1 12096.098,E2 12096.098} C_VEL
LIN {X 0,Y 566.765,Z 869.381,A -85,B 0,C 180,E1 12100.636,E2 12100.636} C_VEL
LIN {X 0,Y 556.098,Z 946.916,A -85,B 0,C 180,E1 12103.519,E2 12103.519} C_VEL
LIN {X 0,Y 542.581,Z 1019.926,A -85,B 0,C 180,E1 12108.101,E2 12108.101} C_VEL
LIN {X 0,Y 529.315,Z 1082.698,A -85,B 0,C 180,E1 12114.03,E2 12114.03} C_VEL
LIN {X 0,Y 517.997,Z 1135.044,A -85,B 0,C 180,E1 12121.369,E2 12121.369} C_VEL
LIN {X 0,Y 513.714,Z 1154.588,A -85,B 0,C 180,E1 12125.134,E2 12125.134} C_VEL
LIN {X 0,Y 503.496,Z 1170.322,A -85,B 0,C 180,E1 12128.527,E2 12128.527} C_VEL
LIN {X 0,Y 500.215,Z 1195.263,A -85,B 0,C 180,E1 12136.855,E2 12136.855} C_VEL
LIN {X 0,Y 498.999,Z 1208.362,A -85,B 0,C 180,E1 12145.641,E2 12145.641} C_VEL
LIN {X 0,Y 498.912,Z 1209.398,A -85,B 0,C 180,E1 12152.612,E2 12152.612} C_VEL
LIN {X 0,Y 499.65,Z 1200.589,A -85,B 0,C 180,E1 12160.491,E2 12160.491} C_VEL
LIN {X 0,Y 502.092,Z 1177.757,A -85,B 0,C 180,E1 12169.403,E2 12169.403} C_VEL
LIN {X 0,Y 508.554,Z 1143.182,A -85,B 0,C 180,E1 12177.528,E2 12177.528} C_VEL
LIN {X 0,Y 519.494,Z 1094.149,A -85,B 0,C 180,E1 12185.04,E2 12185.04} C_VEL
LIN {X 0,Y 533.392,Z 1032.396,A -85,B 0,C 180,E1 12191.406,E2 12191.406} C_VEL
LIN {X 0,Y 547.771,Z 961.51,A -85,B 0,C 180,E1 12196.292,E2 12196.292} C_VEL
LIN {X 0,Y 559.351,Z 884.463,A -85,B 0,C 180,E1 12199.559,E2 12199.559} C_VEL
LIN {X 0,Y 559.878,Z 867.519,A -85,B 0,C 180,E1 12200.199,E2 12200.199} C_VEL
LIN {X 0,Y 530.892,Z 811.356,A -85,B 0,C 180,E1 12205.674,E2 12205.674} C_VEL
LIN {X 0,Y 499.931,Z 767.252,A -85,B 0,C 180,E1 12212.092,E2 12212.092} C_VEL
LIN {X 0,Y 497.939,Z 762.06,A -85,B 0,C 180,E1 12212.772,E2 12212.772} C_VEL
LIN {X 0,Y 498.106,Z 762.06,A -85,B 0,C 180,E1 12223.155,E2 12223.155} C_VEL
LIN {X 0,Y 498.383,Z 762.06,A -85,B 0,C 180,E1 12232.105,E2 12232.105} C_VEL
LIN {X 0,Y 498.704,Z 762.06,A -85,B 0,C 180,E1 12239.11,E2 12239.11} C_VEL
LIN {X 0,Y 498.405,Z 762.06,A -85,B 0,C 180,E1 12247.859,E2 12247.859} C_VEL
LIN {X 0,Y 498.023,Z 762.06,A -85,B 0,C 180,E1 12256.811,E2 12256.811} C_VEL
LIN {X 0,Y 497.761,Z 762.06,A -85,B 0,C 180,E1 12266.221,E2 12266.221} C_VEL
LIN {X 0,Y 498.217,Z 763.816,A -85,B 0,C 180,E1 12271.246,E2 12271.246} C_VEL
LIN {X 0,Y 535.181,Z 817.467,A -85,B 0,C 180,E1 12278.817,E2 12278.817} C_VEL
LIN {X 0,Y 559.973,Z 864.644,A -85,B 0,C 180,E1 12283.371,E2 12283.371} C_VEL
LIN {X 0,Y 549.8,Z 939.468,A -85,B 0,C 180,E1 12286.071,E2 12286.071} C_VEL
LIN {X 0,Y 536.271,Z 1006.085,A -85,B 0,C 180,E1 12290.231,E2 12290.231} C_VEL
LIN {X 0,Y 521.894,Z 1064.842,A -85,B 0,C 180,E1 12295.951,E2 12295.951} C_VEL
LIN {X 0,Y 509.627,Z 1113.957,A -85,B 0,C 180,E1 12303.243,E2 12303.243} C_VEL
LIN {X 0,Y 502.436,Z 1149.711,A -85,B 0,C 180,E1 12311.525,E2 12311.525} C_VEL
LIN {X 0,Y 499.756,Z 1172.183,A -85,B 0,C 180,E1 12320.394,E2 12320.394} C_VEL
LIN {X 0,Y 498.974,Z 1179.831,A -85,B 0,C 180,E1 12327.389,E2 12327.389} C_VEL
LIN {X 0,Y 499.097,Z 1178.728,A -85,B 0,C 180,E1 12334.358,E2 12334.358} C_VEL
LIN {X 0,Y 500.514,Z 1164.819,A -85,B 0,C 180,E1 12343.137,E2 12343.137} C_VEL
LIN {X 0,Y 504.895,Z 1135.869,A -85,B 0,C 180,E1 12352.054,E2 12352.054} C_VEL
LIN {X 0,Y 514.234,Z 1094.939,A -85,B 0,C 180,E1 12359.858,E2 12359.858} C_VEL
LIN {X 0,Y 527.847,Z 1041.549,A -85,B 0,C 180,E1 12366.513,E2 12366.513} C_VEL
LIN {X 0,Y 542.22,Z 979.063,A -85,B 0,C 180,E1 12371.615,E2 12371.615} C_VEL
LIN {X 0,Y 554.648,Z 908.721,A -85,B 0,C 180,E1 12375.17,E2 12375.17} C_VEL
LIN {X 0,Y 559.203,Z 861.547,A -85,B 0,C 180,E1 12376.735,E2 12376.735} C_VEL
LIN {X 0,Y 527.232,Z 805.668,A -85,B 0,C 180,E1 12382.505,E2 12382.505} C_VEL
LIN {X 0,Y 497.877,Z 762.06,A -85,B 0,C 180,E1 12389.012,E2 12389.012} C_VEL
LIN {X 0,Y 498.084,Z 762.06,A -85,B 0,C 180,E1 12398.227,E2 12398.227} C_VEL
LIN {X 0,Y 498.928,Z 762.06,A -85,B 0,C 180,E1 12408.613,E2 12408.613} C_VEL
LIN {X 0,Y 498.688,Z 762.06,A -85,B 0,C 180,E1 12419.146,E2 12419.146} C_VEL
LIN {X 0,Y 498.391,Z 762.06,A -85,B 0,C 180,E1 12427.895,E2 12427.895} C_VEL
LIN {X 0,Y 498.043,Z 762.06,A -85,B 0,C 180,E1 12436.848,E2 12436.848} C_VEL
LIN {X 0,Y 497.739,Z 762.06,A -85,B 0,C 180,E1 12446.262,E2 12446.262} C_VEL
LIN {X 0,Y 498.048,Z 764.17,A -85,B 0,C 180,E1 12447.462,E2 12447.462} C_VEL
LIN {X 0,Y 532.953,Z 815.372,A -85,B 0,C 180,E1 12454.729,E2 12454.729} C_VEL
LIN {X 0,Y 561.143,Z 871.111,A -85,B 0,C 180,E1 12460.08,E2 12460.08} C_VEL
LIN {X 0,Y 549.905,Z 949.202,A -85,B 0,C 180,E1 12463.043,E2 12463.043} C_VEL
LIN {X 0,Y 535.897,Z 1020.915,A -85,B 0,C 180,E1 12467.642,E2 12467.642} C_VEL
LIN {X 0,Y 521.61,Z 1085.453,A -85,B 0,C 180,E1 12473.909,E2 12473.909} C_VEL
LIN {X 0,Y 510.353,Z 1135.643,A -85,B 0,C 180,E1 12481.113,E2 12481.113} C_VEL
LIN {X 0,Y 503.496,Z 1170.322,A -85,B 0,C 180,E1 12488.527,E2 12488.527} C_VEL
LIN {X 0,Y 493.33,Z 1183.634,A -85,B 0,C 180,E1 12492.142,E2 12492.142} C_VEL
LIN {X 0,Y 491.257,Z 1202.146,A -85,B 0,C 180,E1 12500.223,E2 12500.223} C_VEL
LIN {X 0,Y 491.102,Z 1209.392,A -85,B 0,C 180,E1 12507.343,E2 12507.343} C_VEL
LIN {X 0,Y 491.264,Z 1206.762,A -85,B 0,C 180,E1 12516.201,E2 12516.201} C_VEL
LIN {X 0,Y 492.114,Z 1192.264,A -85,B 0,C 180,E1 12524.681,E2 12524.681} C_VEL
LIN {X 0,Y 496.652,Z 1164.469,A -85,B 0,C 180,E1 12533.362,E2 12533.362} C_VEL
LIN {X 0,Y 506.001,Z 1121.529,A -85,B 0,C 180,E1 12541.631,E2 12541.631} C_VEL
LIN {X 0,Y 519.027,Z 1066.207,A -85,B 0,C 180,E1 12548.729,E2 12548.729} C_VEL
LIN {X 0,Y 534.461,Z 998.64,A -85,B 0,C 180,E1 12554.574,E2 12554.574} C_VEL
LIN {X 0,Y 548.074,Z 927.853,A -85,B 0,C 180,E1 12558.525,E2 12558.525} C_VEL
LIN {X 0,Y 554.298,Z 871.311,A -85,B 0,C 180,E1 12560.699,E2 12560.699} C_VEL
LIN {X 0,Y 526.762,Z 816.777,A -85,B 0,C 180,E1 12566.156,E2 12566.156} C_VEL
LIN {X 0,Y 493.933,Z 768.998,A -85,B 0,C 180,E1 12573.274,E2 12573.274} C_VEL
LIN {X 0,Y 489.869,Z 762.06,A -85,B 0,C 180,E1 12574.413,E2 12574.413} C_VEL
LIN {X 0,Y 490.138,Z 762.06,A -85,B 0,C 180,E1 12584.72,E2 12584.72} C_VEL
LIN {X 0,Y 490.437,Z 762.06,A -85,B 0,C 180,E1 12593.763,E2 12593.763} C_VEL
LIN {X 0,Y 490.588,Z 762.06,A -85,B 0,C 180,E1 12600.868,E2 12600.868} C_VEL
LIN {X 0,Y 490.338,Z 762.06,A -85,B 0,C 180,E1 12609.784,E2 12609.784} C_VEL
LIN {X 0,Y 489.938,Z 762.06,A -85,B 0,C 180,E1 12619.259,E2 12619.259} C_VEL
LIN {X 0,Y 490.091,Z 763.624,A -85,B 0,C 180,E1 12629.501,E2 12629.501} C_VEL
LIN {X 0,Y 523.591,Z 811.413,A -85,B 0,C 180,E1 12636.955,E2 12636.955} C_VEL
LIN {X 0,Y 554.492,Z 866.567,A -85,B 0,C 180,E1 12642.795,E2 12642.795} C_VEL
LIN {X 0,Y 544.053,Z 940.261,A -85,B 0,C 180,E1 12645.493,E2 12645.493} C_VEL
LIN {X 0,Y 529.874,Z 1007.433,A -85,B 0,C 180,E1 12649.737,E2 12649.737} C_VEL
LIN {X 0,Y 514.709,Z 1066.894,A -85,B 0,C 180,E1 12655.636,E2 12655.636} C_VEL
LIN {X 0,Y 501.91,Z 1115.781,A -85,B 0,C 180,E1 12663.099,E2 12663.099} C_VEL
LIN {X 0,Y 494.642,Z 1150.116,A -85,B 0,C 180,E1 12671.223,E2 12671.223} C_VEL
LIN {X 0,Y 491.785,Z 1172.469,A -85,B 0,C 180,E1 12680.237,E2 12680.237} C_VEL
LIN {X 0,Y 491.007,Z 1180.08,A -85,B 0,C 180,E1 12687.346,E2 12687.346} C_VEL
LIN {X 0,Y 491.125,Z 1178.985,A -85,B 0,C 180,E1 12694.429,E2 12694.429} C_VEL
LIN {X 0,Y 492.606,Z 1165.149,A -85,B 0,C 180,E1 12703.351,E2 12703.351} C_VEL
LIN {X 0,Y 497.281,Z 1136.307,A -85,B 0,C 180,E1 12712.41,E2 12712.41} C_VEL
LIN {X 0,Y 507.446,Z 1093.987,A -85,B 0,C 180,E1 12720.536,E2 12720.536} C_VEL
LIN {X 0,Y 521.74,Z 1040.296,A -85,B 0,C 180,E1 12727.226,E2 12727.226} C_VEL
LIN {X 0,Y 536.908,Z 976.499,A -85,B 0,C 180,E1 12732.379,E2 12732.379} C_VEL
LIN {X 0,Y 549.628,Z 905.473,A -85,B 0,C 180,E1 12735.91,E2 12735.91} C_VEL
LIN {X 0,Y 553.609,Z 865.14,A -85,B 0,C 180,E1 12737.266,E2 12737.266} C_VEL
LIN {X 0,Y 523.214,Z 811.169,A -85,B 0,C 180,E1 12743.002,E2 12743.002} C_VEL
LIN {X 0,Y 492.552,Z 768.003,A -85,B 0,C 180,E1 12749.705,E2 12749.705} C_VEL
LIN {X 0,Y 489.862,Z 762.06,A -85,B 0,C 180,E1 12750.546,E2 12750.546} C_VEL
LIN {X 0,Y 490.091,Z 762.06,A -85,B 0,C 180,E1 12760.701,E2 12760.701} C_VEL
LIN {X 0,Y 490.906,Z 762.06,A -85,B 0,C 180,E1 12768.425,E2 12768.425} C_VEL
LIN {X 0,Y 490.708,Z 762.06,A -85,B 0,C 180,E1 12779.132,E2 12779.132} C_VEL
LIN {X 0,Y 490.373,Z 762.06,A -85,B 0,C 180,E1 12788.025,E2 12788.025} C_VEL
LIN {X 0,Y 489.999,Z 762.06,A -85,B 0,C 180,E1 12797.133,E2 12797.133} C_VEL
LIN {X 0,Y 489.905,Z 763.581,A -85,B 0,C 180,E1 12805.71,E2 12805.71} C_VEL
LIN {X 0,Y 524.42,Z 813.61,A -85,B 0,C 180,E1 12813.42,E2 12813.42} C_VEL
LIN {X 0,Y 553.308,Z 869.252,A -85,B 0,C 180,E1 12819.11,E2 12819.11} C_VEL
LIN {X 0,Y 554.797,Z 879.78,A -85,B 0,C 180,E1 12819.723,E2 12819.723} C_VEL
LIN {X 0,Y 542.944,Z 955.776,A -85,B 0,C 180,E1 12822.798,E2 12822.798} C_VEL
LIN {X 0,Y 528.165,Z 1026.677,A -85,B 0,C 180,E1 12827.563,E2 12827.563} C_VEL
LIN {X 0,Y 513.387,Z 1090.282,A -85,B 0,C 180,E1 12834.038,E2 12834.038} C_VEL
LIN {X 0,Y 501.883,Z 1140.148,A -85,B 0,C 180,E1 12841.566,E2 12841.566} C_VEL
LIN {X 0,Y 494.921,Z 1176.207,A -85,B 0,C 180,E1 12849.834,E2 12849.834} C_VEL
LIN {X 0,Y 493.33,Z 1183.634,A -85,B 0,C 180,E1 12852.142,E2 12852.142} C_VEL
LIN {X 0,Y 484.384,Z 1194.307,A -85,B 0,C 180,E1 12855.973,E2 12855.973} C_VEL
LIN {X 0,Y 483.362,Z 1206.754,A -85,B 0,C 180,E1 12863.694,E2 12863.694} C_VEL
LIN {X 0,Y 483.033,Z 1209.837,A -85,B 0,C 180,E1 12870.898,E2 12870.898} C_VEL
LIN {X 0,Y 483.316,Z 1203.482,A -85,B 0,C 180,E1 12879.023,E2 12879.023} C_VEL
LIN {X 0,Y 485.858,Z 1183.349,A -85,B 0,C 180,E1 12888.243,E2 12888.243} C_VEL
LIN {X 0,Y 492.303,Z 1149.229,A -85,B 0,C 180,E1 12897.022,E2 12897.022} C_VEL
LIN {X 0,Y 503.353,Z 1101.98,A -85,B 0,C 180,E1 12904.902,E2 12904.902} C_VEL
LIN {X 0,Y 518.799,Z 1039.633,A -85,B 0,C 180,E1 12911.875,E2 12911.875} C_VEL
LIN {X 0,Y 534.524,Z 969.467,A -85,B 0,C 180,E1 12917.059,E2 12917.059} C_VEL
LIN {X 0,Y 547.648,Z 892.422,A -85,B 0,C 180,E1 12920.539,E2 12920.539} C_VEL
LIN {X 0,Y 548.428,Z 874.426,A -85,B 0,C 180,E1 12921.275,E2 12921.275} C_VEL
LIN {X 0,Y 522.421,Z 821.747,A -85,B 0,C 180,E1 12926.68,E2 12926.68} C_VEL
LIN {X 0,Y 490.9,Z 775.848,A -85,B 0,C 180,E1 12933.715,E2 12933.715} C_VEL
LIN {X 0,Y 481.8,Z 762.06,A -85,B 0,C 180,E1 12936.478,E2 12936.478} C_VEL
LIN {X 0,Y 482.217,Z 762.06,A -85,B 0,C 180,E1 12946.327,E2 12946.327} C_VEL
LIN {X 0,Y 483.132,Z 762.06,A -85,B 0,C 180,E1 12957.281,E2 12957.281} C_VEL
LIN {X 0,Y 482.662,Z 762.06,A -85,B 0,C 180,E1 12966.3,E2 12966.3} C_VEL
LIN {X 0,Y 482.01,Z 762.06,A -85,B 0,C 180,E1 12976.348,E2 12976.348} C_VEL
LIN {X 0,Y 481.697,Z 762.06,A -85,B 0,C 180,E1 12986.204,E2 12986.204} C_VEL
LIN {X 0,Y 482.107,Z 764.247,A -85,B 0,C 180,E1 12987.645,E2 12987.645} C_VEL
LIN {X 0,Y 511.61,Z 804.776,A -85,B 0,C 180,E1 12994.83,E2 12994.83} C_VEL
LIN {X 0,Y 542.596,Z 857.094,A -85,B 0,C 180,E1 13000.945,E2 13000.945} C_VEL
LIN {X 0,Y 548.724,Z 872.052,A -85,B 0,C 180,E1 13002.302,E2 13002.302} C_VEL
LIN {X 0,Y 537.507,Z 945.562,A -85,B 0,C 180,E1 13005.118,E2 13005.118} C_VEL
LIN {X 0,Y 522.626,Z 1012.222,A -85,B 0,C 180,E1 13009.511,E2 13009.511} C_VEL
LIN {X 0,Y 507.141,Z 1070.115,A -85,B 0,C 180,E1 13015.481,E2 13015.481} C_VEL
LIN {X 0,Y 494.005,Z 1118.354,A -85,B 0,C 180,E1 13023.102,E2 13023.102} C_VEL
LIN {X 0,Y 486.592,Z 1152.605,A -85,B 0,C 180,E1 13031.575,E2 13031.575} C_VEL
LIN {X 0,Y 483.836,Z 1172.756,A -85,B 0,C 180,E1 13040.075,E2 13040.075} C_VEL
LIN {X 0,Y 483.015,Z 1180.33,A -85,B 0,C 180,E1 13047.302,E2 13047.302} C_VEL
LIN {X 0,Y 483.133,Z 1179.242,A -85,B 0,C 180,E1 13054.503,E2 13054.503} C_VEL
LIN {X 0,Y 484.407,Z 1167.467,A -85,B 0,C 180,E1 13062.661,E2 13062.661} C_VEL
LIN {X 0,Y 489.066,Z 1140.203,A -85,B 0,C 180,E1 13071.905,E2 13071.905} C_VEL
LIN {X 0,Y 498.947,Z 1100.023,A -85,B 0,C 180,E1 13080.102,E2 13080.102} C_VEL
LIN {X 0,Y 513.397,Z 1047.528,A -85,B 0,C 180,E1 13087.052,E2 13087.052} C_VEL
LIN {X 0,Y 528.847,Z 986.021,A -85,B 0,C 180,E1 13092.37,E2 13092.37} C_VEL
LIN {X 0,Y 542.772,Z 915.356,A -85,B 0,C 180,E1 13096.156,E2 13096.156} C_VEL
LIN {X 0,Y 547.923,Z 868.518,A -85,B 0,C 180,E1 13097.833,E2 13097.833} C_VEL
LIN {X 0,Y 518.38,Z 815.061,A -85,B 0,C 180,E1 13103.682,E2 13103.682} C_VEL
LIN {X 0,Y 485.954,Z 769.047,A -85,B 0,C 180,E1 13111.152,E2 13111.152} C_VEL
LIN {X 0,Y 481.84,Z 762.06,A -85,B 0,C 180,E1 13112.843,E2 13112.843} C_VEL
LIN {X 0,Y 482.368,Z 762.06,A -85,B 0,C 180,E1 13123.52,E2 13123.52} C_VEL
LIN {X 0,Y 482.465,Z 762.06,A -85,B 0,C 180,E1 13131.954,E2 13131.954} C_VEL
LIN {X 0,Y 482.709,Z 762.06,A -85,B 0,C 180,E1 13139.118,E2 13139.118} C_VEL
LIN {X 0,Y 482.374,Z 762.06,A -85,B 0,C 180,E1 13148.159,E2 13148.159} C_VEL
LIN {X 0,Y 481.975,Z 762.06,A -85,B 0,C 180,E1 13157.427,E2 13157.427} C_VEL
LIN {X 0,Y 482.028,Z 764.082,A -85,B 0,C 180,E1 13163.884,E2 13163.884} C_VEL
LIN {X 0,Y 513.533,Z 808.308,A -85,B 0,C 180,E1 13171.539,E2 13171.539} C_VEL
LIN {X 0,Y 542.48,Z 860.594,A -85,B 0,C 180,E1 13177.442,E2 13177.442} C_VEL
LIN {X 0,Y 549.342,Z 880.594,A -85,B 0,C 180,E1 13179.123,E2 13179.123} C_VEL
LIN {X 0,Y 537.098,Z 956.246,A -85,B 0,C 180,E1 13182.212,E2 13182.212} C_VEL
LIN {X 0,Y 521.688,Z 1027.231,A -85,B 0,C 180,E1 13187.036,E2 13187.036} C_VEL
LIN {X 0,Y 506.048,Z 1091.4,A -85,B 0,C 180,E1 13193.709,E2 13193.709} C_VEL
LIN {X 0,Y 494.197,Z 1140.831,A -85,B 0,C 180,E1 13201.319,E2 13201.319} C_VEL
LIN {X 0,Y 486.874,Z 1177.741,A -85,B 0,C 180,E1 13209.961,E2 13209.961} C_VEL
LIN {X 0,Y 484.384,Z 1194.307,A -85,B 0,C 180,E1 13215.973,E2 13215.973} C_VEL
LIN {X 0,Y 475.312,Z 1202.253,A -85,B 0,C 180,E1 13219.97,E2 13219.97} C_VEL
LIN {X 0,Y 475.084,Z 1209.386,A -85,B 0,C 180,E1 13227.254,E2 13227.254} C_VEL
LIN {X 0,Y 475.201,Z 1208.357,A -85,B 0,C 180,E1 13234.574,E2 13234.574} C_VEL
LIN {X 0,Y 475.881,Z 1196.307,A -85,B 0,C 180,E1 13243.317,E2 13243.317} C_VEL
LIN {X 0,Y 479.126,Z 1174.233,A -85,B 0,C 180,E1 13251.344,E2 13251.344} C_VEL
LIN {X 0,Y 487.001,Z 1137.986,A -85,B 0,C 180,E1 13259.608,E2 13259.608} C_VEL
LIN {X 0,Y 499.857,Z 1087.357,A -85,B 0,C 180,E1 13267.308,E2 13267.308} C_VEL
LIN {X 0,Y 516.37,Z 1023.725,A -85,B 0,C 180,E1 13273.848,E2 13273.848} C_VEL
LIN {X 0,Y 531.88,Z 954.715,A -85,B 0,C 180,E1 13278.483,E2 13278.483} C_VEL
LIN {X 0,Y 542.906,Z 878.351,A -85,B 0,C 180,E1 13281.769,E2 13281.769} C_VEL
LIN {X 0,Y 518.501,Z 827.504,A -85,B 0,C 180,E1 13287.129,E2 13287.129} C_VEL
LIN {X 0,Y 488.192,Z 782.737,A -85,B 0,C 180,E1 13294.094,E2 13294.094} C_VEL
LIN {X 0,Y 473.86,Z 762.06,A -85,B 0,C 180,E1 13298.612,E2 13298.612} C_VEL
LIN {X 0,Y 474.357,Z 762.06,A -85,B 0,C 180,E1 13307.977,E2 13307.977} C_VEL
LIN {X 0,Y 475.132,Z 762.06,A -85,B 0,C 180,E1 13317.235,E2 13317.235} C_VEL
LIN {X 0,Y 474.63,Z 762.06,A -85,B 0,C 180,E1 13326.407,E2 13326.407} C_VEL
LIN {X 0,Y 474.069,Z 762.06,A -85,B 0,C 180,E1 13335.772,E2 13335.772} C_VEL
LIN {X 0,Y 473.922,Z 763.962,A -85,B 0,C 180,E1 13345.499,E2 13345.499} C_VEL
LIN {X 0,Y 503.163,Z 803.099,A -85,B 0,C 180,E1 13353.271,E2 13353.271} C_VEL
LIN {X 0,Y 535.052,Z 856.241,A -85,B 0,C 180,E1 13359.905,E2 13359.905} C_VEL
LIN {X 0,Y 543.119,Z 876.135,A -85,B 0,C 180,E1 13361.767,E2 13361.767} C_VEL
LIN {X 0,Y 531.067,Z 949.635,A -85,B 0,C 180,E1 13364.689,E2 13364.689} C_VEL
LIN {X 0,Y 515.477,Z 1016.426,A -85,B 0,C 180,E1 13369.253,E2 13369.253} C_VEL
LIN {X 0,Y 499.094,Z 1075.115,A -85,B 0,C 180,E1 13375.561,E2 13375.561} C_VEL
LIN {X 0,Y 485.906,Z 1122.074,A -85,B 0,C 180,E1 13383.345,E2 13383.345} C_VEL
LIN {X 0,Y 478.444,Z 1155.575,A -85,B 0,C 180,E1 13392.121,E2 13392.121} C_VEL
LIN {X 0,Y 475.595,Z 1174.955,A -85,B 0,C 180,E1 13401.12,E2 13401.12} C_VEL
LIN {X 0,Y 474.981,Z 1181.068,A -85,B 0,C 180,E1 13409.087,E2 13409.087} C_VEL
LIN {X 0,Y 475.513,Z 1176.794,A -85,B 0,C 180,E1 13417.331,E2 13417.331} C_VEL
LIN {X 0,Y 477.221,Z 1160.156,A -85,B 0,C 180,E1 13426.146,E2 13426.146} C_VEL
LIN {X 0,Y 483.434,Z 1130.908,A -85,B 0,C 180,E1 13434.643,E2 13434.643} C_VEL
LIN {X 0,Y 495.381,Z 1087.457,A -85,B 0,C 180,E1 13442.62,E2 13442.62} C_VEL
LIN {X 0,Y 511.497,Z 1031.085,A -85,B 0,C 180,E1 13449.329,E2 13449.329} C_VEL
LIN {X 0,Y 527.385,Z 967.741,A -85,B 0,C 180,E1 13454.168,E2 13454.168} C_VEL
LIN {X 0,Y 540.397,Z 896.553,A -85,B 0,C 180,E1 13457.493,E2 13457.493} C_VEL
LIN {X 0,Y 542.463,Z 872.238,A -85,B 0,C 180,E1 13458.376,E2 13458.376} C_VEL
LIN {X 0,Y 513.57,Z 819.206,A -85,B 0,C 180,E1 13464.376,E2 13464.376} C_VEL
LIN {X 0,Y 482.969,Z 775.848,A -85,B 0,C 180,E1 13471.64,E2 13471.64} C_VEL
LIN {X 0,Y 473.853,Z 762.06,A -85,B 0,C 180,E1 13474.775,E2 13474.775} C_VEL
LIN {X 0,Y 474.475,Z 762.06,A -85,B 0,C 180,E1 13484.242,E2 13484.242} C_VEL
LIN {X 0,Y 474.446,Z 762.06,A -85,B 0,C 180,E1 13493.59,E2 13493.59} C_VEL
LIN {X 0,Y 474.485,Z 762.06,A -85,B 0,C 180,E1 13500.935,E2 13500.935} C_VEL
LIN {X 0,Y 474.292,Z 762.06,A -85,B 0,C 180,E1 13510.156,E2 13510.156} C_VEL
LIN {X 0,Y 473.872,Z 762.06,A -85,B 0,C 180,E1 13519.672,E2 13519.672} C_VEL
LIN {X 0,Y 474.077,Z 764.125,A -85,B 0,C 180,E1 13521.824,E2 13521.824} C_VEL
LIN {X 0,Y 503.279,Z 804.323,A -85,B 0,C 180,E1 13529.624,E2 13529.624} C_VEL
LIN {X 0,Y 532.873,Z 855.005,A -85,B 0,C 180,E1 13535.936,E2 13535.936} C_VEL
LIN {X 0,Y 543.727,Z 883.261,A -85,B 0,C 180,E1 13538.57,E2 13538.57} C_VEL
LIN {X 0,Y 531.06,Z 958.027,A -85,B 0,C 180,E1 13541.685,E2 13541.685} C_VEL
LIN {X 0,Y 514.883,Z 1029.406,A -85,B 0,C 180,E1 13546.633,E2 13546.633} C_VEL
LIN {X 0,Y 499.176,Z 1090.778,A -85,B 0,C 180,E1 13553.141,E2 13553.141} C_VEL
LIN {X 0,Y 486.467,Z 1141.691,A -85,B 0,C 180,E1 13561.104,E2 13561.104} C_VEL
LIN {X 0,Y 478.685,Z 1179.373,A -85,B 0,C 180,E1 13570.199,E2 13570.199} C_VEL
LIN {X 0,Y 475.554,Z 1200.574,A -85,B 0,C 180,E1 13578.967,E2 13578.967} C_VEL
LIN {X 0,Y 475.312,Z 1202.253,A -85,B 0,C 180,E1 13579.97,E2 13579.97} C_VEL
LIN {X 0,Y 467.2,Z 1207.319,A -85,B 0,C 180,E1 13584.141,E2 13584.141} C_VEL
LIN {X 0,Y 467.037,Z 1209.836,A -85,B 0,C 180,E1 13590.928,E2 13590.928} C_VEL
LIN {X 0,Y 467.387,Z 1203.475,A -85,B 0,C 180,E1 13599.335,E2 13599.335} C_VEL
LIN {X 0,Y 469.936,Z 1184.42,A -85,B 0,C 180,E1 13608.337,E2 13608.337} C_VEL
LIN {X 0,Y 476.9,Z 1149.447,A -85,B 0,C 180,E1 13617.695,E2 13617.695} C_VEL
LIN {X 0,Y 489.516,Z 1100.234,A -85,B 0,C 180,E1 13626.112,E2 13626.112} C_VEL
LIN {X 0,Y 506.234,Z 1039.043,A -85,B 0,C 180,E1 13633.107,E2 13633.107} C_VEL
LIN {X 0,Y 523.001,Z 969.793,A -85,B 0,C 180,E1 13638.294,E2 13638.294} C_VEL
LIN {X 0,Y 536.945,Z 893.207,A -85,B 0,C 180,E1 13641.806,E2 13641.806} C_VEL
LIN {X 0,Y 536.866,Z 880.742,A -85,B 0,C 180,E1 13642.418,E2 13642.418} C_VEL
LIN {X 0,Y 513.693,Z 831.567,A -85,B 0,C 180,E1 13647.787,E2 13647.787} C_VEL
LIN {X 0,Y 484.204,Z 788.129,A -85,B 0,C 180,E1 13654.823,E2 13654.823} C_VEL
LIN {X 0,Y 465.996,Z 762.06,A -85,B 0,C 180,E1 13660.833,E2 13660.833} C_VEL
LIN {X 0,Y 466.379,Z 762.06,A -85,B 0,C 180,E1 13671.559,E2 13671.559} C_VEL
LIN {X 0,Y 466.737,Z 762.06,A -85,B 0,C 180,E1 13679.049,E2 13679.049} C_VEL
LIN {X 0,Y 466.352,Z 762.06,A -85,B 0,C 180,E1 13688.402,E2 13688.402} C_VEL
LIN {X 0,Y 465.894,Z 762.06,A -85,B 0,C 180,E1 13698.009,E2 13698.009} C_VEL
LIN {X 0,Y 465.878,Z 763.87,A -85,B 0,C 180,E1 13703.12,E2 13703.12} C_VEL
LIN {X 0,Y 492.858,Z 799.519,A -85,B 0,C 180,E1 13711.145,E2 13711.145} C_VEL
LIN {X 0,Y 523.873,Z 848.605,A -85,B 0,C 180,E1 13718.045,E2 13718.045} C_VEL
LIN {X 0,Y 537.477,Z 879.816,A -85,B 0,C 180,E1 13721.217,E2 13721.217} C_VEL
LIN {X 0,Y 524.871,Z 952.902,A -85,B 0,C 180,E1 13724.214,E2 13724.214} C_VEL
LIN {X 0,Y 508.713,Z 1019.336,A -85,B 0,C 180,E1 13728.878,E2 13728.878} C_VEL
LIN {X 0,Y 491.877,Z 1077.025,A -85,B 0,C 180,E1 13735.226,E2 13735.226} C_VEL
LIN {X 0,Y 478.246,Z 1123.557,A -85,B 0,C 180,E1 13743.139,E2 13743.139} C_VEL
LIN {X 0,Y 470.483,Z 1156.837,A -85,B 0,C 180,E1 13752.171,E2 13752.171} C_VEL
LIN {X 0,Y 467.5,Z 1176.026,A -85,B 0,C 180,E1 13761.608,E2 13761.608} C_VEL
LIN {X 0,Y 466.984,Z 1181.315,A -85,B 0,C 180,E1 13769.071,E2 13769.071} C_VEL
LIN {X 0,Y 467.442,Z 1178.101,A -85,B 0,C 180,E1 13776.522,E2 13776.522} C_VEL
LIN {X 0,Y 469.085,Z 1162.819,A -85,B 0,C 180,E1 13785.471,E2 13785.471} C_VEL
LIN {X 0,Y 474.834,Z 1135.405,A -85,B 0,C 180,E1 13794.046,E2 13794.046} C_VEL
LIN {X 0,Y 486.726,Z 1093.653,A -85,B 0,C 180,E1 13802.249,E2 13802.249} C_VEL
LIN {X 0,Y 503.045,Z 1039.55,A -85,B 0,C 180,E1 13809.122,E2 13809.122} C_VEL
LIN {X 0,Y 519.813,Z 976.211,A -85,B 0,C 180,E1 13814.291,E2 13814.291} C_VEL
LIN {X 0,Y 533.637,Z 905.772,A -85,B 0,C 180,E1 13817.834,E2 13817.834} C_VEL
LIN {X 0,Y 537.007,Z 875.948,A -85,B 0,C 180,E1 13818.93,E2 13818.93} C_VEL
LIN {X 0,Y 509.292,Z 824.191,A -85,B 0,C 180,E1 13824.962,E2 13824.962} C_VEL
LIN {X 0,Y 479.872,Z 782.299,A -85,B 0,C 180,E1 13832.184,E2 13832.184} C_VEL
LIN {X 0,Y 465.851,Z 762.06,A -85,B 0,C 180,E1 13837.006,E2 13837.006} C_VEL
LIN {X 0,Y 466.837,Z 762.06,A -85,B 0,C 180,E1 13847.819,E2 13847.819} C_VEL
LIN {X 0,Y 466.726,Z 762.06,A -85,B 0,C 180,E1 13859.087,E2 13859.087} C_VEL
LIN {X 0,Y 466.348,Z 762.06,A -85,B 0,C 180,E1 13868.441,E2 13868.441} C_VEL
LIN {X 0,Y 465.901,Z 762.06,A -85,B 0,C 180,E1 13878.774,E2 13878.774} C_VEL
LIN {X 0,Y 472.194,Z 772.477,A -85,B 0,C 180,E1 13881.621,E2 13881.621} C_VEL
LIN {X 0,Y 499.4,Z 809.457,A -85,B 0,C 180,E1 13889.038,E2 13889.038} C_VEL
LIN {X 0,Y 528.195,Z 860.095,A -85,B 0,C 180,E1 13895.501,E2 13895.501} C_VEL
LIN {X 0,Y 538.037,Z 886.725,A -85,B 0,C 180,E1 13898.027,E2 13898.027} C_VEL
LIN {X 0,Y 525.004,Z 960.123,A -85,B 0,C 180,E1 13901.161,E2 13901.161} C_VEL
LIN {X 0,Y 508.469,Z 1030.17,A -85,B 0,C 180,E1 13906.095,E2 13906.095} C_VEL
LIN {X 0,Y 491.849,Z 1092.351,A -85,B 0,C 180,E1 13912.822,E2 13912.822} C_VEL
LIN {X 0,Y 478.502,Z 1143.811,A -85,B 0,C 180,E1 13921.129,E2 13921.129} C_VEL
LIN {X 0,Y 470.671,Z 1180.227,A -85,B 0,C 180,E1 13930.224,E2 13930.224} C_VEL
LIN {X 0,Y 467.628,Z 1200.571,A -85,B 0,C 180,E1 13938.778,E2 13938.778} C_VEL
LIN {X 0,Y 467.2,Z 1207.319,A -85,B 0,C 180,E1 13944.141,E2 13944.141} C_VEL
LIN {X 0,Y 459.298,Z 1209.68,A -85,B 0,C 180,E1 13948.405,E2 13948.405} C_VEL
LIN {X 0,Y 459.22,Z 1206.738,A -85,B 0,C 180,E1 13956.635,E2 13956.635} C_VEL
LIN {X 0,Y 460.618,Z 1191.633,A -85,B 0,C 180,E1 13965.759,E2 13965.759} C_VEL
LIN {X 0,Y 466.313,Z 1162.66,A -85,B 0,C 180,E1 13975.008,E2 13975.008} C_VEL
LIN {X 0,Y 477.448,Z 1119.006,A -85,B 0,C 180,E1 13983.767,E2 13983.767} C_VEL
LIN {X 0,Y 493.451,Z 1062.397,A -85,B 0,C 180,E1 13991.355,E2 13991.355} C_VEL
LIN {X 0,Y 511.129,Z 996.108,A -85,B 0,C 180,E1 13997.227,E2 13997.227} C_VEL
LIN {X 0,Y 526.805,Z 924.303,A -85,B 0,C 180,E1 14001.236,E2 14001.236} C_VEL
LIN {X 0,Y 531.44,Z 884.625,A -85,B 0,C 180,E1 14002.937,E2 14002.937} C_VEL
LIN {X 0,Y 509.408,Z 836.695,A -85,B 0,C 180,E1 14008.333,E2 14008.333} C_VEL
LIN {X 0,Y 480.783,Z 793.842,A -85,B 0,C 180,E1 14015.439,E2 14015.439} C_VEL
LIN {X 0,Y 460.693,Z 768.049,A -85,B 0,C 180,E1 14022.175,E2 14022.175} C_VEL
LIN {X 0,Y 458.011,Z 762.06,A -85,B 0,C 180,E1 14023.619,E2 14023.619} C_VEL
LIN {X 0,Y 458.392,Z 762.06,A -85,B 0,C 180,E1 14033.325,E2 14033.325} C_VEL
LIN {X 0,Y 458.607,Z 762.06,A -85,B 0,C 180,E1 14040.929,E2 14040.929} C_VEL
LIN {X 0,Y 458.284,Z 762.06,A -85,B 0,C 180,E1 14050.476,E2 14050.476} C_VEL
LIN {X 0,Y 457.975,Z 763.698,A -85,B 0,C 180,E1 14060.401,E2 14060.401} C_VEL
LIN {X 0,Y 482.389,Z 795.777,A -85,B 0,C 180,E1 14068.725,E2 14068.725} C_VEL
LIN {X 0,Y 511.632,Z 839.487,A -85,B 0,C 180,E1 14075.78,E2 14075.78} C_VEL
LIN {X 0,Y 532.079,Z 882.458,A -85,B 0,C 180,E1 14080.631,E2 14080.631} C_VEL
LIN {X 0,Y 518.7,Z 956.459,A -85,B 0,C 180,E1 14083.751,E2 14083.751} C_VEL
LIN {X 0,Y 501.914,Z 1022.243,A -85,B 0,C 180,E1 14088.486,E2 14088.486} C_VEL
LIN {X 0,Y 484.652,Z 1079.093,A -85,B 0,C 180,E1 14094.905,E2 14094.905} C_VEL
LIN {X 0,Y 470.494,Z 1125.171,A -85,B 0,C 180,E1 14102.979,E2 14102.979} C_VEL
LIN {X 0,Y 462.435,Z 1158.43,A -85,B 0,C 180,E1 14112.349,E2 14112.349} C_VEL
LIN {X 0,Y 459.533,Z 1176.291,A -85,B 0,C 180,E1 14121.462,E2 14121.462} C_VEL
LIN {X 0,Y 458.987,Z 1181.563,A -85,B 0,C 180,E1 14129.055,E2 14129.055} C_VEL
LIN {X 0,Y 459.462,Z 1177.635,A -85,B 0,C 180,E1 14137.341,E2 14137.341} C_VEL
LIN {X 0,Y 461.535,Z 1160.906,A -85,B 0,C 180,E1 14146.653,E2 14146.653} C_VEL
LIN {X 0,Y 468.762,Z 1130.818,A -85,B 0,C 180,E1 14155.648,E2 14155.648} C_VEL
LIN {X 0,Y 482.199,Z 1086.401,A -85,B 0,C 180,E1 14163.936,E2 14163.936} C_VEL
LIN {X 0,Y 499.67,Z 1029.657,A -85,B 0,C 180,E1 14170.735,E2 14170.735} C_VEL
LIN {X 0,Y 516.512,Z 966.661,A -85,B 0,C 180,E1 14175.544,E2 14175.544} C_VEL
LIN {X 0,Y 530.169,Z 895.963,A -85,B 0,C 180,E1 14178.839,E2 14178.839} C_VEL
LIN {X 0,Y 531.207,Z 878.783,A -85,B 0,C 180,E1 14179.566,E2 14179.566} C_VEL
LIN {X 0,Y 503.956,Z 827.23,A -85,B 0,C 180,E1 14185.812,E2 14185.812} C_VEL
LIN {X 0,Y 473.967,Z 784.016,A -85,B 0,C 180,E1 14193.637,E2 14193.637} C_VEL
LIN {X 0,Y 457.974,Z 762.06,A -85,B 0,C 180,E1 14199.656,E2 14199.656} C_VEL
LIN {X 0,Y 458.718,Z 762.06,A -85,B 0,C 180,E1 14209.534,E2 14209.534} C_VEL
LIN {X 0,Y 458.727,Z 762.06,A -85,B 0,C 180,E1 14219.072,E2 14219.072} C_VEL
LIN {X 0,Y 458.324,Z 762.06,A -85,B 0,C 180,E1 14228.59,E2 14228.59} C_VEL
LIN {X 0,Y 458.153,Z 763.969,A -85,B 0,C 180,E1 14236.786,E2 14236.786} C_VEL
LIN {X 0,Y 480.435,Z 793.582,A -85,B 0,C 180,E1 14244.504,E2 14244.504} C_VEL
LIN {X 0,Y 509.626,Z 837.721,A -85,B 0,C 180,E1 14251.762,E2 14251.762} C_VEL
LIN {X 0,Y 532.633,Z 887.552,A -85,B 0,C 180,E1 14257.373,E2 14257.373} C_VEL
LIN {X 0,Y 518.896,Z 962.657,A -85,B 0,C 180,E1 14260.648,E2 14260.648} C_VEL
LIN {X 0,Y 501.755,Z 1032.271,A -85,B 0,C 180,E1 14265.658,E2 14265.658} C_VEL
LIN {X 0,Y 484.728,Z 1093.29,A -85,B 0,C 180,E1 14272.403,E2 14272.403} C_VEL
LIN {X 0,Y 470.752,Z 1144.604,A -85,B 0,C 180,E1 14280.906,E2 14280.906} C_VEL
LIN {X 0,Y 462.547,Z 1181.297,A -85,B 0,C 180,E1 14290.361,E2 14290.361} C_VEL
LIN {X 0,Y 459.416,Z 1201.974,A -85,B 0,C 180,E1 14299.538,E2 14299.538} C_VEL
LIN {X 0,Y 459.298,Z 1209.68,A -85,B 0,C 180,E1 14308.405,E2 14308.405} C_VEL
LIN {X 0,Y 450.951,Z 1209.223,A -85,B 0,C 180,E1 14312.758,E2 14312.758} C_VEL
LIN {X 0,Y 451.821,Z 1200.088,A -85,B 0,C 180,E1 14321.616,E2 14321.616} C_VEL
LIN {X 0,Y 454.919,Z 1178.395,A -85,B 0,C 180,E1 14330.833,E2 14330.833} C_VEL
LIN {X 0,Y 463.197,Z 1143.722,A -85,B 0,C 180,E1 14339.694,E2 14339.694} C_VEL
LIN {X 0,Y 477.854,Z 1092.87,A -85,B 0,C 180,E1 14348.23,E2 14348.23} C_VEL
LIN {X 0,Y 496.025,Z 1031.153,A -85,B 0,C 180,E1 14355.073,E2 14355.073} C_VEL
LIN {X 0,Y 513.677,Z 961.868,A -85,B 0,C 180,E1 14360.055,E2 14360.055} C_VEL
LIN {X 0,Y 525.989,Z 888.323,A -85,B 0,C 180,E1 14363.485,E2 14363.485} C_VEL
LIN {X 0,Y 505.112,Z 841.848,A -85,B 0,C 180,E1 14368.864,E2 14368.864} C_VEL
LIN {X 0,Y 476.637,Z 798.111,A -85,B 0,C 180,E1 14376.309,E2 14376.309} C_VEL
LIN {X 0,Y 454.797,Z 769.386,A -85,B 0,C 180,E1 14384.297,E2 14384.297} C_VEL
LIN {X 0,Y 450.296,Z 762.06,A -85,B 0,C 180,E1 14387.324,E2 14387.324} C_VEL
LIN {X 0,Y 451.067,Z 762.06,A -85,B 0,C 180,E1 14397.087,E2 14397.087} C_VEL
LIN {X 0,Y 450.546,Z 762.06,A -85,B 0,C 180,E1 14406.823,E2 14406.823} C_VEL
LIN {X 0,Y 449.953,Z 763.138,A -85,B 0,C 180,E1 14417.02,E2 14417.02} C_VEL
LIN {X 0,Y 472.467,Z 792.45,A -85,B 0,C 180,E1 14426.123,E2 14426.123} C_VEL
LIN {X 0,Y 500.202,Z 832.662,A -85,B 0,C 180,E1 14433.553,E2 14433.553} C_VEL
LIN {X 0,Y 526.336,Z 883.417,A -85,B 0,C 180,E1 14439.892,E2 14439.892} C_VEL
LIN {X 0,Y 513.154,Z 957.023,A -85,B 0,C 180,E1 14443.1,E2 14443.1} C_VEL
LIN {X 0,Y 495.862,Z 1022.661,A -85,B 0,C 180,E1 14447.864,E2 14447.864} C_VEL
LIN {X 0,Y 477.93,Z 1079.447,A -85,B 0,C 180,E1 14454.337,E2 14454.337} C_VEL
LIN {X 0,Y 463.084,Z 1125.653,A -85,B 0,C 180,E1 14462.555,E2 14462.555} C_VEL
LIN {X 0,Y 454.673,Z 1158.614,A -85,B 0,C 180,E1 14471.999,E2 14471.999} C_VEL
LIN {X 0,Y 451.568,Z 1176.549,A -85,B 0,C 180,E1 14481.31,E2 14481.31} C_VEL
LIN {X 0,Y 450.99,Z 1181.81,A -85,B 0,C 180,E1 14489.039,E2 14489.039} C_VEL
LIN {X 0,Y 451.494,Z 1177.819,A -85,B 0,C 180,E1 14497.534,E2 14497.534} C_VEL
LIN {X 0,Y 453.523,Z 1162.284,A -85,B 0,C 180,E1 14506.515,E2 14506.515} C_VEL
LIN {X 0,Y 460.623,Z 1133.606,A -85,B 0,C 180,E1 14515.503,E2 14515.503} C_VEL
LIN {X 0,Y 474.371,Z 1089.867,A -85,B 0,C 180,E1 14524.02,E2 14524.02} C_VEL
LIN {X 0,Y 492.35,Z 1033.873,A -85,B 0,C 180,E1 14530.978,E2 14530.978} C_VEL
LIN {X 0,Y 510.165,Z 970.078,A -85,B 0,C 180,E1 14536.011,E2 14536.011} C_VEL
LIN {X 0,Y 524.502,Z 899.49,A -85,B 0,C 180,E1 14539.397,E2 14539.397} C_VEL
LIN {X 0,Y 525.785,Z 882.559,A -85,B 0,C 180,E1 14540.125,E2 14540.125} C_VEL
LIN {X 0,Y 499.765,Z 832.307,A -85,B 0,C 180,E1 14546.423,E2 14546.423} C_VEL
LIN {X 0,Y 471.388,Z 790.992,A -85,B 0,C 180,E1 14554.084,E2 14554.084} C_VEL
LIN {X 0,Y 453.16,Z 768.384,A -85,B 0,C 180,E1 14561.091,E2 14561.091} C_VEL
LIN {X 0,Y 450.297,Z 762.06,A -85,B 0,C 180,E1 14563.372,E2 14563.372} C_VEL
LIN {X 0,Y 450.479,Z 762.06,A -85,B 0,C 180,E1 14571.299,E2 14571.299} C_VEL
LIN {X 0,Y 450.728,Z 762.06,A -85,B 0,C 180,E1 14579.055,E2 14579.055} C_VEL
LIN {X 0,Y 450.323,Z 762.06,A -85,B 0,C 180,E1 14588.744,E2 14588.744} C_VEL
LIN {X 0,Y 450.383,Z 763.885,A -85,B 0,C 180,E1 14593.603,E2 14593.603} C_VEL
LIN {X 0,Y 468.546,Z 788.072,A -85,B 0,C 180,E1 14601.196,E2 14601.196} C_VEL
LIN {X 0,Y 494.433,Z 824.687,A -85,B 0,C 180,E1 14608.556,E2 14608.556} C_VEL
LIN {X 0,Y 520.278,Z 873.404,A -85,B 0,C 180,E1 14614.947,E2 14614.947} C_VEL
LIN {X 0,Y 526.692,Z 894.659,A -85,B 0,C 180,E1 14616.949,E2 14616.949} C_VEL
LIN {X 0,Y 512.31,Z 967.802,A -85,B 0,C 180,E1 14620.275,E2 14620.275} C_VEL
LIN {X 0,Y 494.538,Z 1036.309,A -85,B 0,C 180,E1 14625.384,E2 14625.384} C_VEL
LIN {X 0,Y 477.07,Z 1096.192,A -85,B 0,C 180,E1 14632.244,E2 14632.244} C_VEL
LIN {X 0,Y 462.748,Z 1146.411,A -85,B 0,C 180,E1 14640.904,E2 14640.904} C_VEL
LIN {X 0,Y 454.438,Z 1182.334,A -85,B 0,C 180,E1 14650.504,E2 14650.504} C_VEL
LIN {X 0,Y 451.453,Z 1201.695,A -85,B 0,C 180,E1 14659.351,E2 14659.351} C_VEL
LIN {X 0,Y 451.304,Z 1209.527,A -85,B 0,C 180,E1 14668.438,E2 14668.438} C_VEL
LIN {X 0,Y 450.951,Z 1209.223,A -85,B 0,C 180,E1 14672.758,E2 14672.758} C_VEL
LIN {X 0,Y 443.218,Z 1205.935,A -85,B 0,C 180,E1 14677.185,E2 14677.185} C_VEL
LIN {X 0,Y 444.916,Z 1190.992,A -85,B 0,C 180,E1 14686.33,E2 14686.33} C_VEL
LIN {X 0,Y 451.568,Z 1160.711,A -85,B 0,C 180,E1 14696.152,E2 14696.152} C_VEL
LIN {X 0,Y 464.236,Z 1115.69,A -85,B 0,C 180,E1 14705.33,E2 14705.33} C_VEL
LIN {X 0,Y 481.755,Z 1058.761,A -85,B 0,C 180,E1 14712.982,E2 14712.982} C_VEL
LIN {X 0,Y 500.852,Z 991.396,A -85,B 0,C 180,E1 14718.894,E2 14718.894} C_VEL
LIN {X 0,Y 517.453,Z 918.472,A -85,B 0,C 180,E1 14722.847,E2 14722.847} C_VEL
LIN {X 0,Y 520.4,Z 891.363,A -85,B 0,C 180,E1 14724.107,E2 14724.107} C_VEL
LIN {X 0,Y 499.865,Z 845.035,A -85,B 0,C 180,E1 14729.666,E2 14729.666} C_VEL
LIN {X 0,Y 473.037,Z 803.966,A -85,B 0,C 180,E1 14737.022,E2 14737.022} C_VEL
LIN {X 0,Y 452.731,Z 776.857,A -85,B 0,C 180,E1 14744.736,E2 14744.736} C_VEL
LIN {X 0,Y 444.668,Z 767.686,A -85,B 0,C 180,E1 14749.159,E2 14749.159} C_VEL
